// TwinCAT 3 PLC project mobject_graph_vision_pack
// Title: mobject-graph-vision-pack
// Company: mobject
// Author: mobject dev team
// ProjectVersion: 0.7.0
// ProgramVersion: 3.1.4024.0
// libraries:
//   mobject-core,0.5.0,mobject
//   mobject-graph,0.14.0,mobject
//   mobject-graph-plc-pack,0.15.0,mobject
//   Tc2_Standard, * (Beckhoff Automation GmbH)
//   Tc2_System, * (Beckhoff Automation GmbH)
//   Tc2_Utilities, * (Beckhoff Automation GmbH)
//   Tc3_Module, * (Beckhoff Automation GmbH)
//   Tc3_Vision, * (Beckhoff Automation GmbH)
// project tree:
//   Datatypes/Aliases/ _GVCP_REGISTER_ADDRESS.TcPOU, _TcVnMatrix2x3_LREAL.TcPOU (not stored), _TcVnArray4_Point2_REAL.TcPOU, _TcVnArray4_LREAL.TcPOU, _TcVnArray33_UDINT.TcPOU (excluded from build), _TcVnArray10_ITcVnImage.TcPOU, _TcVnArray3_Point2_REAL.TcPOU, _TcVnArray7_LREAL.TcPOU, _TcVnArray8_LREAL.TcPOU, _TcVnMatrix3x3_LREAL.TcPOU, _TcVnPoint.TcPOU, _TcVnPoint2_LREAL.TcPOU, _TcVnPoint3_REAL.TcPOU, _TcVnPoint3_LREAL.TcPOU, _TcVnPoint2_REAL.TcPOU, _TcVnRectangle.TcPOU, _TcVnVector2_DINT.TcPOU, _TcVnPoint2_DINT.TcPOU, _ALIASTYP.TcPOU (excluded from build), _TcVnVector2_INT.TcPOU, _TcVnVector3_SINT.TcPOU, _TcVnVector3_INT.TcPOU, _TcVnVector2_SINT.TcPOU, _TcVnVector2_LREAL.TcPOU, _TcVnVector2_UINT.TcPOU, _TcVnVector2_USINT.TcPOU, _TcVnVector3_UINT.TcPOU, _TcVnVector3_USINT.TcPOU, _TcVnVector4_INT.TcPOU, _TcVnVector4_SINT.TcPOU, _TcVnVector4_LREAL.TcPOU, _TcVnVector3_REAL.TcPOU, _TcVnVector3_LREAL.TcPOU, _TcVnVector2_REAL.TcPOU, _TcVnVector4_DINT.TcPOU, _TcVnVector4_UINT.TcPOU, _TcVnVector4_USINT.TcPOU
//   Datatypes/Arrays/ _Array0to1OfARRAYTYP.TcPOU (excluded from build), _Array0to1OfDINT.TcPOU, _Array0to1OfINT.TcPOU, _Array0to1OfLREAL.TcPOU, _Array0to1OfREAL.TcPOU, _Array0to1OfSINT.TcPOU, _Array0to1OfUINT.TcPOU, _Array0to1OfUSINT.TcPOU, _Array0to1_0to2OfLREAL.TcPOU, _Array0to2_0to2OfLREAL.TcPOU, _Array0to2OfINT.TcPOU, _Array0to2OfLREAL.TcPOU, _Array0to2OfREAL.TcPOU, _Array0to2OfSINT.TcPOU, _Array0to2OfTcVnPoint2_REAL.TcPOU, _Array0to2OfUINT.TcPOU, _Array0to2OfUSINT.TcPOU, _Array0to32OfUDINT.TcPOU, _Array0to3OfDINT.TcPOU, _Array0to3OfINT.TcPOU, _Array0to3OfLREAL.TcPOU, _Array0to3OfSINT.TcPOU, _Array0to3OfTcVnPoint2_REAL.TcPOU, _Array0to3OfUINT.TcPOU, _Array0to3OfUSINT.TcPOU, _Array0to6OfLREAL.TcPOU, _Array0to7OfLREAL.TcPOU, _Array0to9OfITcVnImage.TcPOU
//   Datatypes/Enums/ _ETcVn2dCodeSearchStrategy.TcPOU, _ETcVnAdaptiveThresholdMethod.TcPOU, _ETcVnBarcodeSearchDirection.TcPOU, _ETcVnBarcodeType.TcPOU, _ETcVnBlobCombination.TcPOU, _ETcVnBorderInterpolationMethod.TcPOU, _ETcVnBoostClassifierType.TcPOU (not stored) (excluded from build), _ETcVnCalibrationPattern.TcPOU, _ETcVnCalibrationPatternOrigin.TcPOU, _ETcVnCameraState.TcPOU, _ETcVnClusteringAlgorithm.TcPOU, _ETcVnColorMap.TcPOU, _ETcVnColorMapSize.TcPOU, _ETcVnColorSpaceTransform.TcPOU, _ETcVnColorTrainingMethod.TcPOU, _ETcVnConnectedComponentsAlgorithm.TcPOU, _ETcVnContainerExportFormat.TcPOU, _ETcVnContourApproximationMethod.TcPOU, _ETcVnContourRetrievalMode.TcPOU, _ETcVnContoursMatchComparisonMethod.TcPOU, _ETcVnDiffusivityTypeKAZE.TcPOU, _ETcVnDistanceTransformationLabel.TcPOU, _ETcVnDistanceTransformationMask.TcPOU, _ETcVnDistanceType.TcPOU, _ETcVnDrawMatchesFlags.TcPOU, _ETcVnDrawShape.TcPOU, _ETcVnEdgeDetectionAlgorithm.TcPOU, _ETcVnEdgeDirection.TcPOU, _ETcVnElementType.TcPOU, _ETcVnEstimationAlgorithm.TcPOU, _ETcVnExtremePointDirection.TcPOU, _ETcVnFeatureDescriptorTypeAKAZE.TcPOU, _ETcVnFeatureScalingType.TcPOU (excluded from build), _ETcVnFeatureScoreTypeORB.TcPOU, _ETcVnFilterDirection.TcPOU, _ETcVnFlipAxis.TcPOU, _ETcVnFontType.TcPOU, _ETcVnHoughMethod.TcPOU, _ETcVnInitializableFunction.TcPOU (excluded from build), _ETcVnInterpolationType.TcPOU, _ETcVnKeypointDetectionTypeAGAST.TcPOU, _ETcVnKeypointDetectionTypeFAST.TcPOU, _ETcVnKnn.TcPOU (excluded from build), _ETcVnLineType.TcPOU, _ETcVnMorphologicalOperator.TcPOU, _ETcVnNbc.TcPOU (excluded from build), _ETcVnNormalizationType.TcPOU, _ETcVnOcrModelType.TcPOU (excluded from build), _ETcVnTimestamp.TcPOU (excluded from build), _ETcVnOcrOptions.TcPOU (excluded from build), _ETcVnOrientationMethod.TcPOU, _ETcVnPaddingMode.TcPOU (excluded from build), _ETcVnPixelConnectivity.TcPOU, _ETcVnPixelEncoding.TcPOU, _ETcVnPixelPackMode.TcPOU, _ETcVnPrototypeClusterer.TcPOU (excluded from build), _ETcVnRectangleIntersection.TcPOU, _ETcVnRotationAngle.TcPOU, _ETcVnRTrees.TcPOU (excluded from build), _ETcVnSignedNormalization.TcPOU, _ETcVnSolvePnPMethod.TcPOU (excluded from build), _ETcVnSta.TcPOU (excluded from build), _ETcVnStructuringElementShape.TcPOU, _ETcVnSvm.TcPOU (excluded from build), _ETcVnSvmKernelType.TcPOU (excluded from build), _ETcVnSvmSgdClassifierMarginType.TcPOU (excluded from build), _ETcVnSvmSgdClassifierType.TcPOU (excluded from build), _ETcVnTemplateMatchMethod.TcPOU, _ETcVnThresholdType.TcPOU, _ETcVnVectorCompareMethod.TcPOU, _ETcVnWorldCoordinateSystem.TcPOU, _ETcWatchdogAccumulationType.TcPOU, _GEV_CAMERA_STATE.TcPOU
//   Datatypes/Interfaces/ _ITcVnContainer.TcPOU, _ITcVnImage.TcPOU
//   Datatypes/Structs/ _TcVnDMatch.TcPOU (not stored), _TcVnKeyPoint.TcPOU, _TcVnImageInfo.TcPOU, _TcVnCodeGrades1D.TcPOU (not stored) (excluded from build), _TcVnParamsMSER.TcPOU (not stored), _TcVnParamsKAZE.TcPOU, _TcVnParamsAKAZE.TcPOU (not stored), _TcVnParamsORB.TcPOU, _TcVnParamsSB.TcPOU (not stored), _TcVnParamsBRISK.TcPOU (not stored), _TcVnParamsFAST.TcPOU, _TcVnParamsBlobDetection.TcPOU, _TcVnParamsAGAST.TcPOU, _TcVnCameraCalibrationOptions.TcPOU (not stored), _TcVnParamsGFTT.TcPOU (not stored), _TcVnRotatedRectangle.TcPOU, _TcVnCircularArc.TcPOU, _TcVnSize2_REAL.TcPOU, _TcVnPixelFormat.TcPOU, _TcVnRectangle_DINT.TcPOU, _TcVnRectangle_UDINT.TcPOU
//   Datatypes/ VisionDatatypePack.TcPOU
//   / GVL_COLOURS.TcGVL, VisionPack.TcPOU
//   Nodes/Algebraic Container Operations/ Node_F_VN_AddToContainerElements_DINT.TcPOU, Node_F_VN_AddToContainerElements_INT.TcPOU, Node_F_VN_AddToContainerElements_LREAL.TcPOU, Node_F_VN_AddToContainerElements_REAL.TcPOU, Node_F_VN_AddToContainerElements_SINT.TcPOU (not stored), Node_F_VN_AddToContainerElements_TcVnKeyPoint.TcPOU, Node_F_VN_AddToContainerElements_TcVnPoint2_DINT.TcPOU, Node_F_VN_AddToContainerElements_TcVnPoint2_LREAL.TcPOU, Node_F_VN_AddToContainerElements_TcVnPoint2_REAL.TcPOU, Node_F_VN_AddToContainerElements_TcVnPoint3_LREAL.TcPOU, Node_F_VN_AddToContainerElements_TcVnPoint3_REAL.TcPOU, Node_F_VN_AddToContainerElements_TcVnRectangle_DINT.TcPOU, Node_F_VN_AddToContainerElements_TcVnVector2_DINT.TcPOU, Node_F_VN_AddToContainerElements_TcVnVector2_INT.TcPOU, Node_F_VN_AddToContainerElements_TcVnVector2_REAL.TcPOU, Node_F_VN_AddToContainerElements_TcVnVector2_SINT.TcPOU, Node_F_VN_AddToContainerElements_TcVnVector2_UINT.TcPOU, Node_F_VN_AddToContainerElements_TcVnVector2_USINT.TcPOU, Node_F_VN_AddToContainerElements_TcVnVector3_INT.TcPOU, Node_F_VN_AddToContainerElements_TcVnVector3_REAL.TcPOU, Node_F_VN_AddToContainerElements_TcVnVector3_SINT.TcPOU, Node_F_VN_AddToContainerElements_TcVnVector3_UINT.TcPOU, Node_F_VN_AddToContainerElements_TcVnVector3_USINT.TcPOU, Node_F_VN_AddToContainerElements_TcVnVector4_DINT.TcPOU, Node_F_VN_AddToContainerElements_TcVnVector4_INT.TcPOU, Node_F_VN_AddToContainerElements_TcVnVector4_LREAL.TcPOU, Node_F_VN_AddToContainerElements_TcVnVector4_SINT.TcPOU, Node_F_VN_AddToContainerElements_TcVnVector4_UINT.TcPOU, Node_F_VN_AddToContainerElements_TcVnVector4_USINT.TcPOU, Node_F_VN_AddToContainerElements_UDINT.TcPOU (not stored), Node_F_VN_AddToContainerElements_UINT.TcPOU (not stored), Node_F_VN_AddToContainerElements_ULINT.TcPOU (not stored), Node_F_VN_AddToContainerElements_USINT.TcPOU (not stored)
//   Nodes/Algebraic Image Operations/ Node_F_VN_AddImages.TcPOU (not stored), Node_F_VN_ElementwiseExp.TcPOU, Node_F_VN_ElementwiseLog.TcPOU (not stored), Node_F_VN_MultiplyImageWithScalar.TcPOU (not stored), Node_F_VN_SubtractScalarFromImage.TcPOU (not stored), Node_F_VN_MultiplyImages.TcPOU, Node_F_VN_SubtractImages.TcPOU (not stored), Node_F_VN_MaxImage.TcPOU (not stored), Node_F_VN_BitwiseOrImages.TcPOU (not stored), Node_F_VN_BitwiseNotImage.TcPOU, Node_F_VN_BitwiseAndImages.TcPOU, Node_F_VN_BitwiseXorImages.TcPOU, Node_F_VN_MinImage.TcPOU (not stored), Node_F_VN_DivideImages.TcPOU, Node_F_VN_SubtractImageFromScalar.TcPOU (not stored), Node_F_VN_AddScalarToImage.TcPOU (not stored)
//   Nodes/Basic Container Operations/ Node_F_VN_AppendToContainer_DINT.TcPOU, Node_F_VN_AppendToContainer_INT.TcPOU, Node_F_VN_AppendToContainer_ITcVnContainer.TcPOU, Node_F_VN_AppendToContainer_ITcVnImage.TcPOU, Node_F_VN_AppendToContainer_LREAL.TcPOU, Node_F_VN_AppendToContainer_REAL.TcPOU, Node_F_VN_AppendToContainer_SINT.TcPOU, Node_F_VN_AppendToContainer_TcVnKeyPoint.TcPOU, Node_F_VN_AppendToContainer_TcVnPoint2_DINT.TcPOU, Node_F_VN_AppendToContainer_TcVnPoint2_LREAL.TcPOU, Node_F_VN_AppendToContainer_TcVnPoint2_REAL.TcPOU, Node_F_VN_AppendToContainer_TcVnPoint3_LREAL.TcPOU, Node_F_VN_AppendToContainer_TcVnPoint3_REAL.TcPOU, Node_F_VN_AppendToContainer_TcVnRectangle_DINT.TcPOU, Node_F_VN_AppendToContainer_TcVnDMatch.TcPOU, Node_F_VN_AppendToContainer_TcVnVector2_DINT.TcPOU, Node_F_VN_AppendToContainer_TcVnVector2_INT.TcPOU, Node_F_VN_AppendToContainer_TcVnVector2_REAL.TcPOU, Node_F_VN_AppendToContainer_TcVnVector2_SINT.TcPOU, Node_F_VN_AppendToContainer_TcVnVector2_UINT.TcPOU, Node_F_VN_AppendToContainer_TcVnVector2_USINT.TcPOU, Node_F_VN_AppendToContainer_TcVnVector3_INT.TcPOU, Node_F_VN_AppendToContainer_TcVnVector3_REAL.TcPOU, Node_F_VN_AppendToContainer_TcVnVector3_SINT.TcPOU, Node_F_VN_AppendToContainer_TcVnVector3_UINT.TcPOU, Node_F_VN_AppendToContainer_TcVnVector3_USINT.TcPOU, Node_F_VN_AppendToContainer_TcVnVector4_DINT.TcPOU, Node_F_VN_AppendToContainer_TcVnVector4_INT.TcPOU, Node_F_VN_AppendToContainer_TcVnVector4_LREAL.TcPOU, Node_F_VN_AppendToContainer_TcVnVector4_SINT.TcPOU, Node_F_VN_AppendToContainer_TcVnVector4_UINT.TcPOU, Node_F_VN_AppendToContainer_TcVnVector4_USINT.TcPOU, Node_F_VN_AppendToContainer_UDINT.TcPOU, Node_F_VN_AppendToContainer_UINT.TcPOU, Node_F_VN_AppendToContainer_ULINT.TcPOU, Node_F_VN_AppendToContainer_USINT.TcPOU, Node_F_VN_FillContainerExp_DINT.TcPOU (not stored), Node_F_VN_FillContainerExp_INT.TcPOU, Node_F_VN_FillContainerExp_ITcVnImage.TcPOU, Node_F_VN_FillContainerExp_LREAL.TcPOU (not stored), Node_F_VN_FillContainerExp_REAL.TcPOU (not stored), Node_F_VN_FillContainerExp_SINT.TcPOU, Node_F_VN_FillContainerExp_TcVnDMatch.TcPOU, Node_F_VN_FillContainerExp_TcVnKeyPoint.TcPOU, Node_F_VN_FillContainerExp_TcVnPoint2_DINT.TcPOU, Node_F_VN_FillContainerExp_TcVnPoint2_LREAL.TcPOU, Node_F_VN_FillContainerExp_TcVnPoint2_REAL.TcPOU, Node_F_VN_FillContainerExp_TcVnPoint3_LREAL.TcPOU, Node_F_VN_FillContainerExp_TcVnPoint3_REAL.TcPOU, Node_F_VN_FillContainerExp_TcVnRectangle_DINT.TcPOU, Node_F_VN_FillContainerExp_TcVnVector2_DINT.TcPOU, Node_F_VN_FillContainerExp_TcVnVector2_INT.TcPOU, Node_F_VN_FillContainerExp_TcVnVector2_REAL.TcPOU, Node_F_VN_FillContainerExp_TcVnVector2_SINT.TcPOU, Node_F_VN_FillContainerExp_TcVnVector2_UINT.TcPOU, Node_F_VN_FillContainerExp_TcVnVector2_USINT.TcPOU, Node_F_VN_FillContainerExp_TcVnVector3_INT.TcPOU, Node_F_VN_FillContainerExp_TcVnVector3_REAL.TcPOU, Node_F_VN_FillContainerExp_TcVnVector3_SINT.TcPOU, Node_F_VN_FillContainerExp_TcVnVector3_UINT.TcPOU, Node_F_VN_FillContainerExp_TcVnVector3_USINT.TcPOU, Node_F_VN_FillContainerExp_TcVnVector4_DINT.TcPOU, Node_F_VN_FillContainerExp_TcVnVector4_INT.TcPOU, Node_F_VN_FillContainerExp_TcVnVector4_LREAL.TcPOU, Node_F_VN_FillContainerExp_TcVnVector4_SINT.TcPOU, Node_F_VN_FillContainerExp_TcVnVector4_UINT.TcPOU, Node_F_VN_FillContainerExp_TcVnVector4_USINT.TcPOU, Node_F_VN_FillContainerExp_UDINT.TcPOU, Node_F_VN_FillContainerExp_UINT.TcPOU, Node_F_VN_FillContainerExp_ULINT.TcPOU (not stored), Node_F_VN_FillContainerExp_USINT.TcPOU, Node_F_VN_FillContainer_DINT.TcPOU, Node_F_VN_FillContainer_INT.TcPOU, Node_F_VN_FillContainer_ITcVnImage.TcPOU, Node_F_VN_FillContainer_LREAL.TcPOU, Node_F_VN_FillContainer_REAL.TcPOU, Node_F_VN_FillContainer_SINT.TcPOU, Node_F_VN_FillContainer_TcVnDMatch.TcPOU, Node_F_VN_FillContainer_TcVnKeyPoint.TcPOU, Node_F_VN_FillContainer_TcVnPoint2_DINT.TcPOU, Node_F_VN_FillContainer_TcVnPoint2_LREAL.TcPOU, Node_F_VN_FillContainer_TcVnPoint2_REAL.TcPOU, Node_F_VN_FillContainer_TcVnPoint3_LREAL.TcPOU, Node_F_VN_FillContainer_TcVnPoint3_REAL.TcPOU, Node_F_VN_FillContainer_TcVnRectangle_DINT.TcPOU, Node_F_VN_FillContainer_TcVnVector2_DINT.TcPOU, Node_F_VN_FillContainer_TcVnVector2_INT.TcPOU, Node_F_VN_FillContainer_TcVnVector2_REAL.TcPOU, Node_F_VN_FillContainer_TcVnVector2_SINT.TcPOU, Node_F_VN_FillContainer_TcVnVector2_UINT.TcPOU, Node_F_VN_FillContainer_TcVnVector2_USINT.TcPOU, Node_F_VN_FillContainer_TcVnVector3_INT.TcPOU, Node_F_VN_FillContainer_TcVnVector3_REAL.TcPOU, Node_F_VN_FillContainer_TcVnVector3_SINT.TcPOU, Node_F_VN_FillContainer_TcVnVector3_UINT.TcPOU, Node_F_VN_FillContainer_TcVnVector3_USINT.TcPOU, Node_F_VN_FillContainer_TcVnVector4_DINT.TcPOU, Node_F_VN_FillContainer_TcVnVector4_INT.TcPOU, Node_F_VN_FillContainer_TcVnVector4_LREAL.TcPOU, Node_F_VN_FillContainer_TcVnVector4_SINT.TcPOU, Node_F_VN_FillContainer_TcVnVector4_UINT.TcPOU, Node_F_VN_FillContainer_TcVnVector4_USINT.TcPOU, Node_F_VN_FillContainer_UDINT.TcPOU, Node_F_VN_FillContainer_UINT.TcPOU, Node_F_VN_FillContainer_ULINT.TcPOU, Node_F_VN_FillContainer_USINT.TcPOU, Node_F_VN_GetAt_DINT.TcPOU (not stored), Node_F_VN_GetAt_INT.TcPOU, Node_F_VN_GetAt_ITcVnContainer.TcPOU (not stored), Node_F_VN_GetAt_ITcVnImage.TcPOU, Node_F_VN_GetAt_LREAL.TcPOU, Node_F_VN_GetAt_REAL.TcPOU (not stored), Node_F_VN_GetAt_SINT.TcPOU (not stored), Node_F_VN_GetAt_TcVnDMatch.TcPOU, Node_F_VN_GetAt_TcVnKeyPoint.TcPOU, Node_F_VN_GetAt_TcVnPoint2_DINT.TcPOU, Node_F_VN_GetAt_TcVnPoint2_LREAL.TcPOU, Node_F_VN_GetAt_TcVnPoint2_REAL.TcPOU, Node_F_VN_GetAt_TcVnPoint3_LREAL.TcPOU, Node_F_VN_GetAt_TcVnPoint3_REAL.TcPOU, Node_F_VN_GetAt_TcVnRectangle_DINT.TcPOU, Node_F_VN_GetAt_TcVnVector2_DINT.TcPOU, Node_F_VN_GetAt_TcVnVector2_INT.TcPOU, Node_F_VN_GetAt_TcVnVector2_REAL.TcPOU, Node_F_VN_GetAt_TcVnVector2_SINT.TcPOU, Node_F_VN_GetAt_TcVnVector2_UINT.TcPOU, Node_F_VN_GetAt_TcVnVector2_USINT.TcPOU, Node_F_VN_GetAt_TcVnVector3_INT.TcPOU, Node_F_VN_GetAt_TcVnVector3_REAL.TcPOU, Node_F_VN_GetAt_TcVnVector3_SINT.TcPOU, Node_F_VN_GetAt_TcVnVector3_UINT.TcPOU, Node_F_VN_GetAt_TcVnVector3_USINT.TcPOU, Node_F_VN_GetAt_TcVnVector4_DINT.TcPOU, Node_F_VN_GetAt_TcVnVector4_INT.TcPOU, Node_F_VN_GetAt_TcVnVector4_LREAL.TcPOU, Node_F_VN_GetAt_TcVnVector4_SINT.TcPOU, Node_F_VN_GetAt_TcVnVector4_UINT.TcPOU, Node_F_VN_GetAt_TcVnVector4_USINT.TcPOU, Node_F_VN_GetAt_UDINT.TcPOU, Node_F_VN_GetAt_UINT.TcPOU (not stored), Node_F_VN_GetAt_ULINT.TcPOU (not stored), Node_F_VN_GetAt_USINT.TcPOU (not stored), Node_F_VN_GetNumberOfElements.TcPOU, Node_F_VN_InsertIntoContainer_DINT.TcPOU, Node_F_VN_InsertIntoContainer_INT.TcPOU, Node_F_VN_InsertIntoContainer_ITcVnContainer.TcPOU, Node_F_VN_InsertIntoContainer_ITcVnImage.TcPOU, Node_F_VN_InsertIntoContainer_LREAL.TcPOU, Node_F_VN_InsertIntoContainer_REAL.TcPOU, Node_F_VN_InsertIntoContainer_SINT.TcPOU, Node_F_VN_InsertIntoContainer_TcVnDMatch.TcPOU, Node_F_VN_InsertIntoContainer_TcVnKeyPoint.TcPOU, Node_F_VN_InsertIntoContainer_TcVnPoint2_DINT.TcPOU, Node_F_VN_InsertIntoContainer_TcVnPoint2_LREAL.TcPOU, Node_F_VN_InsertIntoContainer_TcVnPoint2_REAL.TcPOU, Node_F_VN_InsertIntoContainer_TcVnPoint3_LREAL.TcPOU, Node_F_VN_InsertIntoContainer_TcVnPoint3_REAL.TcPOU, Node_F_VN_InsertIntoContainer_TcVnRectangle_DINT.TcPOU, Node_F_VN_InsertIntoContainer_TcVnVector2_DINT.TcPOU, Node_F_VN_InsertIntoContainer_TcVnVector2_INT.TcPOU, Node_F_VN_InsertIntoContainer_TcVnVector2_REAL.TcPOU, Node_F_VN_InsertIntoContainer_TcVnVector2_SINT.TcPOU, Node_F_VN_InsertIntoContainer_TcVnVector2_UINT.TcPOU, Node_F_VN_InsertIntoContainer_TcVnVector2_USINT.TcPOU, Node_F_VN_InsertIntoContainer_TcVnVector3_INT.TcPOU, Node_F_VN_InsertIntoContainer_TcVnVector3_REAL.TcPOU, Node_F_VN_InsertIntoContainer_TcVnVector3_SINT.TcPOU, Node_F_VN_InsertIntoContainer_TcVnVector3_UINT.TcPOU, Node_F_VN_InsertIntoContainer_TcVnVector3_USINT.TcPOU, Node_F_VN_InsertIntoContainer_TcVnVector4_DINT.TcPOU, Node_F_VN_InsertIntoContainer_TcVnVector4_INT.TcPOU, Node_F_VN_InsertIntoContainer_TcVnVector4_LREAL.TcPOU, Node_F_VN_InsertIntoContainer_TcVnVector4_SINT.TcPOU, Node_F_VN_InsertIntoContainer_TcVnVector4_UINT.TcPOU, Node_F_VN_InsertIntoContainer_TcVnVector4_USINT.TcPOU, Node_F_VN_InsertIntoContainer_UDINT.TcPOU, Node_F_VN_InsertIntoContainer_UINT.TcPOU, Node_F_VN_InsertIntoContainer_ULINT.TcPOU, Node_F_VN_InsertIntoContainer_USINT.TcPOU, Node_F_VN_SetAt_DINT.TcPOU, Node_F_VN_SetAt_INT.TcPOU, Node_F_VN_SetAt_ITcVnContainer.TcPOU, Node_F_VN_SetAt_ITcVnImage.TcPOU, Node_F_VN_SetAt_LREAL.TcPOU, Node_F_VN_SetAt_REAL.TcPOU, Node_F_VN_SetAt_SINT.TcPOU, Node_F_VN_SetAt_TcVnDMatch.TcPOU, Node_F_VN_SetAt_TcVnKeyPoint.TcPOU, Node_F_VN_SetAt_TcVnPoint2_DINT.TcPOU, Node_F_VN_SetAt_TcVnPoint2_LREAL.TcPOU, Node_F_VN_SetAt_TcVnPoint2_REAL.TcPOU, Node_F_VN_SetAt_TcVnPoint3_LREAL.TcPOU, Node_F_VN_SetAt_TcVnPoint3_REAL.TcPOU, Node_F_VN_SetAt_TcVnRectangle_DINT.TcPOU, Node_F_VN_SetAt_TcVnVector2_DINT.TcPOU, Node_F_VN_SetAt_TcVnVector2_INT.TcPOU, Node_F_VN_SetAt_TcVnVector2_REAL.TcPOU, Node_F_VN_SetAt_TcVnVector2_SINT.TcPOU, Node_F_VN_SetAt_TcVnVector2_UINT.TcPOU, Node_F_VN_SetAt_TcVnVector2_USINT.TcPOU, Node_F_VN_SetAt_TcVnVector3_INT.TcPOU, Node_F_VN_SetAt_TcVnVector3_REAL.TcPOU, Node_F_VN_SetAt_TcVnVector3_SINT.TcPOU, Node_F_VN_SetAt_TcVnVector3_UINT.TcPOU, Node_F_VN_SetAt_TcVnVector3_USINT.TcPOU, Node_F_VN_SetAt_TcVnVector4_DINT.TcPOU, Node_F_VN_SetAt_TcVnVector4_INT.TcPOU, Node_F_VN_SetAt_TcVnVector4_LREAL.TcPOU, Node_F_VN_SetAt_TcVnVector4_SINT.TcPOU, Node_F_VN_SetAt_TcVnVector4_UINT.TcPOU, Node_F_VN_SetAt_TcVnVector4_USINT.TcPOU, Node_F_VN_SetAt_UDINT.TcPOU, Node_F_VN_SetAt_UINT.TcPOU, Node_F_VN_SetAt_ULINT.TcPOU, Node_F_VN_SetAt_USINT.TcPOU
//   Nodes/Basic Image Operations/ Node_F_VN_ConvertElementType.TcPOU, Node_F_VN_ConvertElementTypeExp.TcPOU (not stored), Node_F_VN_CopyImage.TcPOU, Node_F_VN_GetPixelFormat.TcPOU, Node_F_VN_ResetRoi.TcPOU (not stored), Node_F_VN_SetRoi.TcPOU (not stored), Node_F_VN_GetImageChannel.TcPOU (not stored), Node_F_VN_GetImageHeight.TcPOU, Node_F_VN_GetImageWidth.TcPOU, Node_F_VN_GetImageInfo.TcPOU, Node_F_VN_GetRoi.TcPOU (not stored), Node_F_VN_SetRoi_TcVnRectangle_DINT.TcPOU (excluded from build)
//   Nodes/Code Reading/ Node_F_VN_ReadQRCode.TcPOU (not stored), Node_F_VN_ReadDataMatrixCode.TcPOU
//   Nodes/Constants/ Node_RGBA_BLUE.TcPOU, Node_RGBA_MAGENTA.TcPOU, Node_RGBA_CYAN.TcPOU, Node_RGBA_YELLOW.TcPOU, Node_RGBA_WHITE.TcPOU, Node_RGBA_RED.TcPOU (not stored), Node_RGBA_GREEN.TcPOU (not stored), Node_RGBA_BLACK.TcPOU (not stored)
//   Nodes/Container Statistics/ Node_F_VN_MaxElementElementwise_DINT.TcPOU, Node_F_VN_MaxElementElementwise_INT.TcPOU, Node_F_VN_MaxElementElementwise_LREAL.TcPOU, Node_F_VN_MaxElementElementwise_REAL.TcPOU, Node_F_VN_MaxElementElementwise_SINT.TcPOU, Node_F_VN_MaxElementElementwise_TcVnPoint2_DINT.TcPOU, Node_F_VN_MaxElementElementwise_TcVnPoint2_LREAL.TcPOU (not stored), Node_F_VN_MaxElementElementwise_TcVnPoint2_REAL.TcPOU (not stored), Node_F_VN_MaxElementElementwise_TcVnPoint3_LREAL.TcPOU (not stored), Node_F_VN_MaxElementElementwise_TcVnPoint3_REAL.TcPOU (not stored), Node_F_VN_MaxElementElementwise_TcVnVector2_DINT.TcPOU (not stored), Node_F_VN_MaxElementElementwise_TcVnVector2_INT.TcPOU (not stored), Node_F_VN_MaxElementElementwise_TcVnVector2_REAL.TcPOU, Node_F_VN_MaxElementElementwise_TcVnVector2_SINT.TcPOU, Node_F_VN_MaxElementElementwise_TcVnVector2_UINT.TcPOU (not stored), Node_F_VN_MaxElementElementwise_TcVnVector2_USINT.TcPOU (not stored), Node_F_VN_MaxElementElementwise_TcVnVector3_INT.TcPOU, Node_F_VN_MaxElementElementwise_TcVnVector3_REAL.TcPOU (not stored), Node_F_VN_MaxElementElementwise_TcVnVector3_SINT.TcPOU, Node_F_VN_MaxElementElementwise_TcVnVector3_UINT.TcPOU (not stored), Node_F_VN_MaxElementElementwise_TcVnVector3_USINT.TcPOU (not stored), Node_F_VN_MaxElementElementwise_TcVnVector4_DINT.TcPOU (not stored), Node_F_VN_MaxElementElementwise_TcVnVector4_INT.TcPOU, Node_F_VN_MaxElementElementwise_TcVnVector4_LREAL.TcPOU (not stored), Node_F_VN_MaxElementElementwise_TcVnVector4_SINT.TcPOU, Node_F_VN_MaxElementElementwise_TcVnVector4_UINT.TcPOU, Node_F_VN_MaxElementElementwise_TcVnVector4_USINT.TcPOU, Node_F_VN_MaxElementElementwise_UDINT.TcPOU, Node_F_VN_MaxElementElementwise_UINT.TcPOU, Node_F_VN_MaxElementElementwise_ULINT.TcPOU, Node_F_VN_MaxElementElementwise_USINT.TcPOU, Node_F_VN_MedianElementElementwise_DINT.TcPOU, Node_F_VN_MedianElementElementwise_INT.TcPOU, Node_F_VN_MedianElementElementwise_LREAL.TcPOU, Node_F_VN_MedianElementElementwise_REAL.TcPOU, Node_F_VN_MedianElementElementwise_SINT.TcPOU, Node_F_VN_MedianElementElementwise_TcVnPoint2_DINT.TcPOU, Node_F_VN_MedianElementElementwise_TcVnPoint2_LREAL.TcPOU, Node_F_VN_MedianElementElementwise_TcVnPoint2_REAL.TcPOU, Node_F_VN_MedianElementElementwise_TcVnPoint3_LREAL.TcPOU, Node_F_VN_MedianElementElementwise_TcVnPoint3_REAL.TcPOU, Node_F_VN_MedianElementElementwise_TcVnVector2_DINT.TcPOU, Node_F_VN_MedianElementElementwise_TcVnVector2_INT.TcPOU, Node_F_VN_MedianElementElementwise_TcVnVector2_REAL.TcPOU, Node_F_VN_MedianElementElementwise_TcVnVector2_SINT.TcPOU, Node_F_VN_MedianElementElementwise_TcVnVector2_UINT.TcPOU, Node_F_VN_MedianElementElementwise_TcVnVector2_USINT.TcPOU, Node_F_VN_MedianElementElementwise_TcVnVector3_INT.TcPOU, Node_F_VN_MedianElementElementwise_TcVnVector3_REAL.TcPOU, Node_F_VN_MedianElementElementwise_TcVnVector3_SINT.TcPOU, Node_F_VN_MedianElementElementwise_TcVnVector3_UINT.TcPOU, Node_F_VN_MedianElementElementwise_TcVnVector3_USINT.TcPOU, Node_F_VN_MedianElementElementwise_TcVnVector4_DINT.TcPOU, Node_F_VN_MedianElementElementwise_TcVnVector4_INT.TcPOU, Node_F_VN_MedianElementElementwise_TcVnVector4_LREAL.TcPOU, Node_F_VN_MedianElementElementwise_TcVnVector4_SINT.TcPOU, Node_F_VN_MedianElementElementwise_TcVnVector4_UINT.TcPOU, Node_F_VN_MedianElementElementwise_TcVnVector4_USINT.TcPOU, Node_F_VN_MedianElementElementwise_UDINT.TcPOU, Node_F_VN_MedianElementElementwise_UINT.TcPOU, Node_F_VN_MedianElementElementwise_ULINT.TcPOU, Node_F_VN_MedianElementElementwise_USINT.TcPOU, Node_F_VN_MinElementElementwise_DINT.TcPOU, Node_F_VN_MinElementElementwise_INT.TcPOU, Node_F_VN_MinElementElementwise_LREAL.TcPOU, Node_F_VN_MinElementElementwise_REAL.TcPOU, Node_F_VN_MinElementElementwise_SINT.TcPOU, Node_F_VN_MinElementElementwise_TcVnPoint2_DINT.TcPOU, Node_F_VN_MinElementElementwise_TcVnPoint2_LREAL.TcPOU, Node_F_VN_MinElementElementwise_TcVnPoint2_REAL.TcPOU, Node_F_VN_MinElementElementwise_TcVnPoint3_LREAL.TcPOU, Node_F_VN_MinElementElementwise_TcVnPoint3_REAL.TcPOU, Node_F_VN_MinElementElementwise_TcVnVector2_DINT.TcPOU, Node_F_VN_MinElementElementwise_TcVnVector2_INT.TcPOU, Node_F_VN_MinElementElementwise_TcVnVector2_REAL.TcPOU, Node_F_VN_MinElementElementwise_TcVnVector2_SINT.TcPOU, Node_F_VN_MinElementElementwise_TcVnVector2_UINT.TcPOU, Node_F_VN_MinElementElementwise_TcVnVector2_USINT.TcPOU, Node_F_VN_MinElementElementwise_TcVnVector3_INT.TcPOU, Node_F_VN_MinElementElementwise_TcVnVector3_REAL.TcPOU, Node_F_VN_MinElementElementwise_TcVnVector3_SINT.TcPOU, Node_F_VN_MinElementElementwise_TcVnVector3_UINT.TcPOU, Node_F_VN_MinElementElementwise_TcVnVector3_USINT.TcPOU, Node_F_VN_MinElementElementwise_TcVnVector4_DINT.TcPOU, Node_F_VN_MinElementElementwise_TcVnVector4_INT.TcPOU, Node_F_VN_MinElementElementwise_TcVnVector4_LREAL.TcPOU, Node_F_VN_MinElementElementwise_TcVnVector4_SINT.TcPOU, Node_F_VN_MinElementElementwise_TcVnVector4_UINT.TcPOU, Node_F_VN_MinElementElementwise_TcVnVector4_USINT.TcPOU, Node_F_VN_MinElementElementwise_UDINT.TcPOU, Node_F_VN_MinElementElementwise_UINT.TcPOU, Node_F_VN_MinElementElementwise_ULINT.TcPOU, Node_F_VN_MinElementElementwise_USINT.TcPOU
//   Nodes/Contour Analysis/ Node_F_VN_FitLine.TcPOU
//   Nodes/Drawing/ Node_F_VN_DrawContours.TcPOU, Node_F_VN_DrawLine.TcPOU, Node_F_VN_DrawCircle.TcPOU (not stored), Node_F_VN_DrawLine_TcVnVector4_LREAL.TcPOU, Node_F_VN_PutLabel.TcPOU, Node_F_VN_PutText.TcPOU
//   Nodes/Geometric and Coordinate Transformations/ Node_F_VN_PyramidDown.TcPOU (not stored), Node_F_VN_FlipImage.TcPOU, Node_F_VN_PyramidUp.TcPOU (not stored)
//   Nodes/Image Analysis/ Node_F_VN_CountNonZeroPixels.TcPOU
//   Nodes/Image Analysis/Object Detection/ Node_F_VN_DetectBlobs.TcPOU
//   Nodes/Image Color and Contrast Processing/ Node_F_VN_ApplyColorMap.TcPOU, Node_F_VN_InvertImageColor.TcPOU (not stored), Node_F_VN_ConvertColorSpace.TcPOU, Node_F_VN_GenerateColorMap.TcPOU, Node_F_VN_NormalizeImage.TcPOU (not stored)
//   Nodes/Image Filtering/ Node_F_VN_LocalMaxima.TcPOU, Node_F_VN_DarkBorderObjects.TcPOU (not stored), Node_F_VN_FillHoles.TcPOU (not stored), Node_F_VN_BoxFilter.TcPOU, Node_F_VN_BrightBorderObjects.TcPOU (not stored), Node_F_VN_GaussianFilter.TcPOU, Node_F_VN_LaplacianFilter.TcPOU, Node_F_VN_LocalMinima.TcPOU (not stored)
//   Nodes/Image Segmentation/ Node_F_VN_Threshold.TcPOU
//   Nodes/Keypoint Features/ Node_F_VN_KeyPointsAGAST.TcPOU (not stored), Node_F_VN_KeyPointsGFTT.TcPOU (not stored), Node_F_VN_KeyPointsFAST.TcPOU (not stored), Node_F_VN_KeyPointsMSER.TcPOU, Node_F_VN_KeyPointsSB.TcPOU (not stored)
//   Nodes/Measurement/ Node_F_VN_LocateEdge.TcPOU, Node_F_VN_LocateEdges.TcPOU (not stored), Node_F_VN_LocateEdgeExp.TcPOU (not stored), Node_F_VN_LocateEdgesExp.TcPOU (not stored), Node_F_VN_LocateEllipse.TcPOU (not stored)
//   Nodes/ VisionNodePack.TcPOU
//   Nodes/VisionNode/ VisionNode.TcPOU (not stored)

// ---- GVL_COLOURS.TcGVL
{attribute 'qualified_only'}
VAR_GLOBAL
    RGBA_BLACK   : TcVnVector4_LREAL := [0, 0, 0, 255];
    RGBA_RED     : TcVnVector4_LREAL := [255, 0, 0, 255];
    RGBA_YELLOW  : TcVnVector4_LREAL := [255, 255, 0, 255];
    RGBA_GREEN   : TcVnVector4_LREAL := [0, 255, 0, 255];
    RGBA_CYAN    : TcVnVector4_LREAL := [0, 255, 255, 255];
    RGBA_BLUE    : TcVnVector4_LREAL := [0, 0, 255, 255];
    RGBA_MAGENTA : TcVnVector4_LREAL := [255, 0, 255, 255];
    RGBA_WHITE   : TcVnVector4_LREAL := [255, 255, 255, 255];
END_VAR

// ---- Datatypes/Aliases/_GVCP_REGISTER_ADDRESS.TcPOU
{attribute 'linkalways'} 
{attribute 'no_explicit_call' := 'This FB is a CLASS and must be accessed using methods or properties'}
{attribute 'enable_dynamic_creation'}
FUNCTION_BLOCK _GVCP_REGISTER_ADDRESS EXTENDS AliasDatatypeBase
VAR
	localData : GVCP_REGISTER_ADDRESS;
	activeData : REFERENCE TO GVCP_REGISTER_ADDRESS REF= localData;
	aliasBaseDatatype : _UDINT(0);
END_VAR

PROPERTY PUBLIC Address : PVOID
GET
Address := ADR(activeData);
END_GET
END_PROPERTY

METHOD PUBLIC ClearReference
VAR_INPUT
END_VAR
activeData REF= localData;
SetBaseDatatypeReference();
END_METHOD

METHOD PUBLIC Clone : I_Datatype
VAR
    pClone : POINTER TO _GVCP_REGISTER_ADDRESS;
END_VAR
pClone := __NEW(_GVCP_REGISTER_ADDRESS);
Clone := pClone^;
END_METHOD

METHOD FB_init : BOOL
VAR_INPUT
	bInitRetains : BOOL; // if TRUE, the retain variables are initialized (warm start / cold start)
	bInCopyCode : BOOL;  // if TRUE, the instance afterwards gets moved into the copy code (online change)
	//InitialValue : TcVnArray33_UDINT; // if possible, not all values can be initialized
END_VAR
//localData := InitialValue; // if possible, not all values can be initialized
SetBaseDatatypeReference();
AddBaseDatatype(aliasBaseDatatype);
END_METHOD

PROPERTY PUBLIC Identifier : T_MAXSTRING
GET
Identifier := 'GVCP_REGISTER_ADDRESS';
END_GET
END_PROPERTY

METHOD PUBLIC MakeReferenceTo
VAR_INPUT
	ReferenceTarget : REFERENCE TO GVCP_REGISTER_ADDRESS;
END_VAR
activeData REF= ReferenceTarget;
SetBaseDatatypeReference();
END_METHOD

METHOD PROTECTED SetBaseDatatypeReference
VAR_INPUT
END_VAR
aliasBaseDatatype.MakeReferenceTo(activeData);
END_METHOD

PROPERTY PUBLIC Size : UDINT
GET
Size := SIZEOF(activeData);
END_GET
END_PROPERTY

METHOD TryMakeReferenceTo : BOOL
VAR_INPUT
	Target : I_Datatype;
END_VAR
VAR
	targetAsAlias : I_AliasDatatype;
	pTargetData : POINTER TO GVCP_REGISTER_ADDRESS;
END_VAR
IF NOT Target.TryResolveAsAliasDatatype(targetAsAlias) THEN
	RETURN;
END_IF

IF targetAsAlias.Identifier <> Identifier THEN
	RETURN;
END_IF

pTargetData := Target.Address;
activeData REF= pTargetData^;
SetBaseDatatypeReference();
TryMakeReferenceTo := TRUE;
END_METHOD

PROPERTY PUBLIC Value : REFERENCE TO GVCP_REGISTER_ADDRESS
GET
Value REF= activeData;
END_GET
END_PROPERTY

END_FUNCTION_BLOCK

// ---- Datatypes/Aliases/_TcVnArray4_Point2_REAL.TcPOU
{attribute 'linkalways'} 
{attribute 'no_explicit_call' := 'This FB is a CLASS and must be accessed using methods or properties'}
{attribute 'enable_dynamic_creation'}
FUNCTION_BLOCK _TcVnArray4_Point2_REAL EXTENDS AliasDatatypeBase
VAR
	localData : TcVnArray4_Point2_REAL;
	activeData : REFERENCE TO TcVnArray4_Point2_REAL REF= localData;
	aliasBaseDatatype : _Array0to3OfTcVnPoint2_REAL;
END_VAR

PROPERTY PUBLIC Address : PVOID
GET
Address := ADR(activeData);
END_GET
END_PROPERTY

METHOD PUBLIC ClearReference
VAR_INPUT
END_VAR
activeData REF= localData;
SetBaseDatatypeReference();
END_METHOD

METHOD PUBLIC Clone : I_Datatype
VAR
    pClone : POINTER TO _TcVnArray4_Point2_REAL;
END_VAR
pClone := __NEW(_TcVnArray4_Point2_REAL);
Clone := pClone^;
END_METHOD

METHOD FB_init : BOOL
VAR_INPUT
	bInitRetains : BOOL; // if TRUE, the retain variables are initialized (warm start / cold start)
	bInCopyCode : BOOL;  // if TRUE, the instance afterwards gets moved into the copy code (online change)
	//InitialValue : TcVnArray4_LREAL; // if possible, not all values can be initialized
END_VAR
//localData := InitialValue; // if possible, not all values can be initialized
SetBaseDatatypeReference();
AddBaseDatatype(aliasBaseDatatype);
END_METHOD

PROPERTY PUBLIC Identifier : T_MAXSTRING
GET
Identifier := 'TcVnArray4_Point2_REAL';
END_GET
END_PROPERTY

METHOD PUBLIC MakeReferenceTo
VAR_INPUT
	ReferenceTarget : REFERENCE TO TcVnArray4_Point2_REAL;
END_VAR
activeData REF= ReferenceTarget;
SetBaseDatatypeReference();
END_METHOD

METHOD PROTECTED SetBaseDatatypeReference
VAR_INPUT
END_VAR
aliasBaseDatatype.MakeReferenceTo(activeData);
END_METHOD

PROPERTY PUBLIC Size : UDINT
GET
Size := SIZEOF(activeData);
END_GET
END_PROPERTY

METHOD TryMakeReferenceTo : BOOL
VAR_INPUT
	Target : I_Datatype;
END_VAR
VAR
	pTargetData : POINTER TO TcVnArray4_Point2_REAL;
END_VAR
IF NOT IsEquivalentTo(Target) THEN
	RETURN;
END_IF

pTargetData := Target.Address;
activeData REF= pTargetData^;
SetBaseDatatypeReference();
TryMakeReferenceTo := TRUE;
END_METHOD

PROPERTY PUBLIC Value : REFERENCE TO TcVnArray4_Point2_REAL
GET
Value REF= activeData;
END_GET
END_PROPERTY

END_FUNCTION_BLOCK

// ---- Datatypes/Arrays/_Array0to3OfTcVnPoint2_REAL.TcPOU
{attribute 'linkalways'} 
{attribute 'no_explicit_call' := 'This FB is a CLASS and must be accessed using methods or properties'}
{attribute 'enable_dynamic_creation'}
FUNCTION_BLOCK _Array0to3OfTcVnPoint2_REAL EXTENDS ArrayDatatypeBase_1D
VAR CONSTANT
	lBound : DINT := 0;
	uBound : DINT := 3;
END_VAR
VAR
	localData : ARRAY [lBound..uBound] OF TcVnPoint2_REAL;
	activeData : REFERENCE TO ARRAY [lBound..uBound] OF TcVnPoint2_REAL REF= localData;
	elements : ARRAY [lBound..uBound] OF _TcVnPoint2_REAL;
	baseType : _TcVnPoint2_REAL;
END_VAR

PROPERTY PUBLIC Address : PVOID
GET
Address := ADR(activeData);
END_GET
END_PROPERTY

PROPERTY PUBLIC BaseDatatype : I_Datatype
GET
BaseDatatype := baseType;
END_GET
END_PROPERTY

METHOD PUBLIC ClearReference
VAR_INPUT
END_VAR
activeData REF= localData;
SetElementReference();
END_METHOD

METHOD PUBLIC Clone : I_Datatype
VAR
    pClone : POINTER TO _Array0to3OfTcVnPoint2_REAL;
END_VAR
pClone := __NEW(_Array0to3OfTcVnPoint2_REAL());
pClone^.Value := Value;
Clone := pClone^;
END_METHOD

METHOD FB_init : BOOL
VAR_INPUT
	bInitRetains : BOOL; // if TRUE, the retain variables are initialized (warm start / cold start)
	bInCopyCode : BOOL;  // if TRUE, the instance afterwards gets moved into the copy code (online change)
END_VAR
SetElementReference();
END_METHOD

METHOD PUBLIC MakeReferenceTo
VAR_INPUT
	ReferenceTarget : REFERENCE TO ARRAY [lBound..uBound] OF TcVnPoint2_REAL;
END_VAR
activeData REF= ReferenceTarget;
SetElementReference();
END_METHOD

METHOD PROTECTED OnSerializeArrayValues
VAR_INPUT
	Serializer : I_Serializer;
END_VAR
VAR
	i : DINT;
END_VAR
FOR i := lBound TO uBound DO
	elements[i].SerializeWith(Serializer);
END_FOR
END_METHOD

METHOD PROTECTED SetElementReference
VAR_INPUT
END_VAR
VAR
	i : DINT;
END_VAR
FOR i := lBound TO uBound DO
	elements[i].MakeReferenceTo(activeData[i]);
END_FOR
END_METHOD

PROPERTY PUBLIC Size : UDINT
GET
Size := SIZEOF(activeData);
END_GET
END_PROPERTY

METHOD PROTECTED TryDeserializeArrayValues : BOOL
VAR_INPUT
	Deserializer : I_Deserializer;
	Feedback : I_DeserializerFeedback;
END_VAR
VAR
	enumerator : I_DeserializerArrayForwardEnumerator;
	i : DINT;
END_VAR
enumerator := Deserializer.GetArrayEnumerator();
i := lBound;

WHILE enumerator.MoveNext() AND i <= uBound DO
	
	IF NOT elements[i].TryDeserializeFrom(enumerator.Current, Feedback) THEN
		EXIT;
	END_IF
	i := i + 1;

END_WHILE
enumerator.Dispose();
END_METHOD

METHOD PUBLIC TryGetElementAsDatatypeByIndex : BOOL
VAR_INPUT
	Index : DINT;
	Destination : REFERENCE TO I_Datatype;
END_VAR
IF Index < lbound OR Index > ubound THEN
	RETURN;
END_IF

Destination := elements[Index];
TryGetElementAsDatatypeByIndex := TRUE;
END_METHOD

METHOD PUBLIC TryGetLowerBound : BOOL
VAR_INPUT
	Dimention : UDINT;
	Destination : REFERENCE TO DINT;
END_VAR
IF Dimention = 1 THEN
	Destination := lBound;
	TryGetLowerBound := TRUE;
END_IF
END_METHOD

METHOD PUBLIC TryGetUpperBound : BOOL
VAR_INPUT
	Dimention : UDINT;
	Destination : REFERENCE TO DINT;
END_VAR
IF Dimention = 1 THEN
	Destination := uBound;
	TryGetUpperBound := TRUE;
END_IF
END_METHOD

METHOD TryMakeReferenceTo : BOOL
VAR_INPUT
	Target : I_Datatype;
END_VAR
VAR
	targetAsArray : I_ArrayDatatype;
	pTargetData : POINTER TO ARRAY [lBound..uBound] OF TcVnPoint2_REAL;
END_VAR
IF NOT Target.TryResolveAsArrayDatatype(targetAsArray) THEN
	RETURN;
END_IF

IF NOT (targetAsArray.Identifier = Identifier) THEN
	RETURN;
END_IF

pTargetData := Target.Address;
activeData REF= pTargetData^;
SetElementReference();
TryMakeReferenceTo := TRUE;
END_METHOD

PROPERTY PUBLIC Value : REFERENCE TO ARRAY [lBound..uBound] OF TcVnPoint2_REAL;
GET
Value ref= activeData;
END_GET
END_PROPERTY

END_FUNCTION_BLOCK

// ---- Datatypes/Aliases/_TcVnPoint2_REAL.TcPOU
{attribute 'linkalways'} 
{attribute 'no_explicit_call' := 'This FB is a CLASS and must be accessed using methods or properties'}
{attribute 'enable_dynamic_creation'}
FUNCTION_BLOCK _TcVnPoint2_REAL EXTENDS AliasDatatypeBase
VAR
	localData : TcVnPoint2_REAL;
	activeData : REFERENCE TO TcVnPoint2_REAL REF= localData;
	aliasBaseDatatype : _TcVnVector2_REAL;
END_VAR

PROPERTY PUBLIC Address : PVOID
GET
Address := ADR(activeData);
END_GET
END_PROPERTY

METHOD PUBLIC ClearReference
VAR_INPUT
END_VAR
activeData REF= localData;
SetBaseDatatypeReference();
END_METHOD

METHOD PUBLIC Clone : I_Datatype
VAR
    pClone : POINTER TO _TcVnPoint2_REAL;
END_VAR
pClone := __NEW(_TcVnPoint2_REAL);
Clone := pClone^;
END_METHOD

METHOD FB_init : BOOL
VAR_INPUT
	bInitRetains : BOOL; // if TRUE, the retain variables are initialized (warm start / cold start)
	bInCopyCode : BOOL;  // if TRUE, the instance afterwards gets moved into the copy code (online change)
	//InitialValue : <type>; // if possible, not all values can be initialized
END_VAR
//localData := InitialValue; // if possible, not all values can be initialized
SetBaseDatatypeReference();
AddBaseDatatype(aliasBaseDatatype);
END_METHOD

PROPERTY PUBLIC Identifier : T_MAXSTRING
GET
Identifier := 'TcVnPoint2_REAL';
END_GET
END_PROPERTY

METHOD PUBLIC MakeReferenceTo
VAR_INPUT
	ReferenceTarget : REFERENCE TO TcVnPoint2_REAL;
END_VAR
activeData REF= ReferenceTarget;
SetBaseDatatypeReference();
END_METHOD

METHOD PROTECTED SetBaseDatatypeReference
VAR_INPUT
END_VAR
aliasBaseDatatype.MakeReferenceTo(activeData);
END_METHOD

PROPERTY PUBLIC Size : UDINT
GET
Size := SIZEOF(activeData);
END_GET
END_PROPERTY

METHOD TryMakeReferenceTo : BOOL
VAR_INPUT
	Target : I_Datatype;
END_VAR
VAR
	pTargetData : POINTER TO TcVnPoint2_REAL;
END_VAR
IF NOT IsEquivalentTo(Target) THEN
	RETURN;
END_IF

pTargetData := Target.Address;
activeData REF= pTargetData^;
SetBaseDatatypeReference();
TryMakeReferenceTo := TRUE;
END_METHOD

PROPERTY PUBLIC Value : REFERENCE TO TcVnPoint2_REAL
GET
Value REF= activeData;
END_GET
END_PROPERTY

END_FUNCTION_BLOCK

// ---- Datatypes/Aliases/_TcVnVector2_REAL.TcPOU
{attribute 'linkalways'} 
{attribute 'no_explicit_call' := 'This FB is a CLASS and must be accessed using methods or properties'}
{attribute 'enable_dynamic_creation'}
FUNCTION_BLOCK _TcVnVector2_REAL EXTENDS AliasDatatypeBase
VAR
	localData : TcVnVector2_REAL;
	activeData : REFERENCE TO TcVnVector2_REAL REF= localData;
	aliasBaseDatatype : _Array0to1OfREAL;
END_VAR

PROPERTY PUBLIC Address : PVOID
GET
Address := ADR(activeData);
END_GET
END_PROPERTY

METHOD PUBLIC ClearReference
VAR_INPUT
END_VAR
activeData REF= localData;
SetBaseDatatypeReference();
END_METHOD

METHOD PUBLIC Clone : I_Datatype
VAR
    pClone : POINTER TO _TcVnVector2_REAL;
END_VAR
pClone := __NEW(_TcVnVector2_REAL);
Clone := pClone^;
END_METHOD

METHOD FB_init : BOOL
VAR_INPUT
	bInitRetains : BOOL; // if TRUE, the retain variables are initialized (warm start / cold start)
	bInCopyCode : BOOL;  // if TRUE, the instance afterwards gets moved into the copy code (online change)
	//InitialValue : <type>; // if possible, not all values can be initialized
END_VAR
//localData := InitialValue; // if possible, not all values can be initialized
SetBaseDatatypeReference();
AddBaseDatatype(aliasBaseDatatype);
END_METHOD

PROPERTY PUBLIC Identifier : T_MAXSTRING
GET
Identifier := 'TcVnVector2_REAL';
END_GET
END_PROPERTY

METHOD PUBLIC MakeReferenceTo
VAR_INPUT
	ReferenceTarget : REFERENCE TO TcVnVector2_REAL;
END_VAR
activeData REF= ReferenceTarget;
SetBaseDatatypeReference();
END_METHOD

METHOD PROTECTED SetBaseDatatypeReference
VAR_INPUT
END_VAR
aliasBaseDatatype.MakeReferenceTo(activeData);
END_METHOD

PROPERTY PUBLIC Size : UDINT
GET
Size := SIZEOF(activeData);
END_GET
END_PROPERTY

METHOD TryMakeReferenceTo : BOOL
VAR_INPUT
	Target : I_Datatype;
END_VAR
VAR
	pTargetData : POINTER TO TcVnVector2_REAL;
END_VAR
IF NOT IsEquivalentTo(Target) THEN
	RETURN;
END_IF

pTargetData := Target.Address;
activeData REF= pTargetData^;
SetBaseDatatypeReference();
TryMakeReferenceTo := TRUE;
END_METHOD

PROPERTY PUBLIC Value : REFERENCE TO TcVnVector2_REAL
GET
Value REF= activeData;
END_GET
END_PROPERTY

END_FUNCTION_BLOCK

// ---- Datatypes/Arrays/_Array0to1OfREAL.TcPOU
{attribute 'linkalways'} 
{attribute 'no_explicit_call' := 'This FB is a CLASS and must be accessed using methods or properties'}
{attribute 'enable_dynamic_creation'}
FUNCTION_BLOCK _Array0to1OfREAL EXTENDS ArrayDatatypeBase_1D
VAR CONSTANT
	lBound : DINT := 0;
	uBound : DINT := 1;
END_VAR
VAR
	localData : ARRAY [lBound..uBound] OF REAL;
	activeData : REFERENCE TO ARRAY [lBound..uBound] OF REAL REF= localData;
	elements : ARRAY [lBound..uBound] OF _REAL(0.0);
	baseType : _REAL(0.0);
END_VAR

PROPERTY PUBLIC Address : PVOID
GET
Address := ADR(activeData);
END_GET
END_PROPERTY

PROPERTY PUBLIC BaseDatatype : I_Datatype
GET
BaseDatatype := baseType;
END_GET
END_PROPERTY

METHOD PUBLIC ClearReference
VAR_INPUT
END_VAR
activeData REF= localData;
SetElementReference();
END_METHOD

METHOD PUBLIC Clone : I_Datatype
VAR
    pClone : POINTER TO _Array0to1OfREAL;
END_VAR
pClone := __NEW(_Array0to1OfREAL());
pClone^.Value := Value;
Clone := pClone^;
END_METHOD

METHOD FB_init : BOOL
VAR_INPUT
	bInitRetains : BOOL; // if TRUE, the retain variables are initialized (warm start / cold start)
	bInCopyCode : BOOL;  // if TRUE, the instance afterwards gets moved into the copy code (online change)
END_VAR
SetElementReference();
END_METHOD

METHOD PUBLIC MakeReferenceTo
VAR_INPUT
	ReferenceTarget : REFERENCE TO ARRAY [lBound..uBound] OF REAL;
END_VAR
activeData REF= ReferenceTarget;
SetElementReference();
END_METHOD

METHOD PROTECTED OnSerializeArrayValues
VAR_INPUT
	Serializer : I_Serializer;
END_VAR
VAR
	i : DINT;
END_VAR
FOR i := lBound TO uBound DO
	elements[i].SerializeWith(Serializer);
END_FOR
END_METHOD

METHOD PROTECTED SetElementReference
VAR_INPUT
END_VAR
VAR
	i : DINT;
END_VAR
FOR i := lBound TO uBound DO
	elements[i].MakeReferenceTo(activeData[i]);
END_FOR
END_METHOD

PROPERTY PUBLIC Size : UDINT
GET
Size := SIZEOF(activeData);
END_GET
END_PROPERTY

METHOD PROTECTED TryDeserializeArrayValues : BOOL
VAR_INPUT
	Deserializer : I_Deserializer;
	Feedback : I_DeserializerFeedback;
END_VAR
VAR
	enumerator : I_DeserializerArrayForwardEnumerator;
	i : DINT;
END_VAR
enumerator := Deserializer.GetArrayEnumerator();
i := lBound;

WHILE enumerator.MoveNext() AND i <= uBound DO
	
	IF NOT elements[i].TryDeserializeFrom(enumerator.Current, Feedback) THEN
		EXIT;
	END_IF
	i := i + 1;

END_WHILE
enumerator.Dispose();
END_METHOD

METHOD PUBLIC TryGetElementAsDatatypeByIndex : BOOL
VAR_INPUT
	Index : DINT;
	Destination : REFERENCE TO I_Datatype;
END_VAR
IF Index < lbound OR Index > ubound THEN
	RETURN;
END_IF

Destination := elements[Index];
TryGetElementAsDatatypeByIndex := TRUE;
END_METHOD

METHOD PUBLIC TryGetLowerBound : BOOL
VAR_INPUT
	Dimention : UDINT;
	Destination : REFERENCE TO DINT;
END_VAR
IF Dimention = 1 THEN
	Destination := lBound;
	TryGetLowerBound := TRUE;
END_IF
END_METHOD

METHOD PUBLIC TryGetUpperBound : BOOL
VAR_INPUT
	Dimention : UDINT;
	Destination : REFERENCE TO DINT;
END_VAR
IF Dimention = 1 THEN
	Destination := uBound;
	TryGetUpperBound := TRUE;
END_IF
END_METHOD

METHOD TryMakeReferenceTo : BOOL
VAR_INPUT
	Target : I_Datatype;
END_VAR
VAR
	pTargetData : POINTER TO ARRAY [lBound..uBound] OF REAL;
END_VAR
IF NOT IsEquivalentTo(Target) THEN
	RETURN;
END_IF

pTargetData := Target.Address;
activeData REF= pTargetData^;
SetElementReference();
TryMakeReferenceTo := TRUE;
END_METHOD

PROPERTY PUBLIC Value : REFERENCE TO ARRAY [lBound..uBound] OF REAL;
GET
Value ref= activeData;
END_GET
END_PROPERTY

END_FUNCTION_BLOCK

// ---- Datatypes/Aliases/_TcVnArray4_LREAL.TcPOU
{attribute 'linkalways'} 
{attribute 'no_explicit_call' := 'This FB is a CLASS and must be accessed using methods or properties'}
{attribute 'enable_dynamic_creation'}
FUNCTION_BLOCK _TcVnArray4_LREAL EXTENDS AliasDatatypeBase
VAR
	localData : TcVnArray4_LREAL;
	activeData : REFERENCE TO TcVnArray4_LREAL REF= localData;
	aliasBaseDatatype : _Array0to3OfLREAL;
END_VAR

PROPERTY PUBLIC Address : PVOID
GET
Address := ADR(activeData);
END_GET
END_PROPERTY

METHOD PUBLIC ClearReference
VAR_INPUT
END_VAR
activeData REF= localData;
SetBaseDatatypeReference();
END_METHOD

METHOD PUBLIC Clone : I_Datatype
VAR
    pClone : POINTER TO _TcVnArray4_LREAL;
END_VAR
pClone := __NEW(_TcVnArray4_LREAL);
Clone := pClone^;
END_METHOD

METHOD FB_init : BOOL
VAR_INPUT
	bInitRetains : BOOL; // if TRUE, the retain variables are initialized (warm start / cold start)
	bInCopyCode : BOOL;  // if TRUE, the instance afterwards gets moved into the copy code (online change)
	//InitialValue : TcVnArray4_LREAL; // if possible, not all values can be initialized
END_VAR
//localData := InitialValue; // if possible, not all values can be initialized
SetBaseDatatypeReference();
AddBaseDatatype(aliasBaseDatatype);
END_METHOD

PROPERTY PUBLIC Identifier : T_MAXSTRING
GET
Identifier := 'TcVnArray4_LREAL';
END_GET
END_PROPERTY

METHOD PUBLIC MakeReferenceTo
VAR_INPUT
	ReferenceTarget : REFERENCE TO TcVnArray4_LREAL;
END_VAR
activeData REF= ReferenceTarget;
SetBaseDatatypeReference();
END_METHOD

METHOD PROTECTED SetBaseDatatypeReference
VAR_INPUT
END_VAR
aliasBaseDatatype.MakeReferenceTo(activeData);
END_METHOD

PROPERTY PUBLIC Size : UDINT
GET
Size := SIZEOF(activeData);
END_GET
END_PROPERTY

METHOD TryMakeReferenceTo : BOOL
VAR_INPUT
	Target : I_Datatype;
END_VAR
VAR
	pTargetData : POINTER TO TcVnArray4_LREAL;
END_VAR
IF NOT IsEquivalentTo(Target) THEN
	RETURN;
END_IF

pTargetData := Target.Address;
activeData REF= pTargetData^;
SetBaseDatatypeReference();
TryMakeReferenceTo := TRUE;
END_METHOD

PROPERTY PUBLIC Value : REFERENCE TO TcVnArray4_LREAL
GET
Value REF= activeData;
END_GET
END_PROPERTY

END_FUNCTION_BLOCK

// ---- Datatypes/Arrays/_Array0to3OfLREAL.TcPOU
{attribute 'linkalways'} 
{attribute 'no_explicit_call' := 'This FB is a CLASS and must be accessed using methods or properties'}
{attribute 'enable_dynamic_creation'}
FUNCTION_BLOCK _Array0to3OfLREAL EXTENDS ArrayDatatypeBase_1D
VAR CONSTANT
	lBound : DINT := 0;
	uBound : DINT := 3;
END_VAR
VAR
	localData : ARRAY [lBound..uBound] OF LREAL;
	activeData : REFERENCE TO ARRAY [lBound..uBound] OF LREAL REF= localData;
	elements : ARRAY [lBound..uBound] OF _LREAL(0.0);
	baseType : _LREAL(0.0);
END_VAR

PROPERTY PUBLIC Address : PVOID
GET
Address := ADR(activeData);
END_GET
END_PROPERTY

PROPERTY PUBLIC BaseDatatype : I_Datatype
GET
BaseDatatype := baseType;
END_GET
END_PROPERTY

METHOD PUBLIC ClearReference
VAR_INPUT
END_VAR
activeData REF= localData;
SetElementReference();
END_METHOD

METHOD PUBLIC Clone : I_Datatype
VAR
    pClone : POINTER TO _Array0to3OfLREAL;
END_VAR
pClone := __NEW(_Array0to3OfLREAL());
pClone^.Value := Value;
Clone := pClone^;
END_METHOD

METHOD FB_init : BOOL
VAR_INPUT
	bInitRetains : BOOL; // if TRUE, the retain variables are initialized (warm start / cold start)
	bInCopyCode : BOOL;  // if TRUE, the instance afterwards gets moved into the copy code (online change)
END_VAR
SetElementReference();
END_METHOD

METHOD PUBLIC MakeReferenceTo
VAR_INPUT
	ReferenceTarget : REFERENCE TO ARRAY [lBound..uBound] OF LREAL;
END_VAR
activeData REF= ReferenceTarget;
SetElementReference();
END_METHOD

METHOD PROTECTED OnSerializeArrayValues
VAR_INPUT
	Serializer : I_Serializer;
END_VAR
VAR
	i : DINT;
END_VAR
FOR i := lBound TO uBound DO
	elements[i].SerializeWith(Serializer);
END_FOR
END_METHOD

METHOD PROTECTED SetElementReference
VAR_INPUT
END_VAR
VAR
	i : DINT;
END_VAR
FOR i := lBound TO uBound DO
	elements[i].MakeReferenceTo(activeData[i]);
END_FOR
END_METHOD

PROPERTY PUBLIC Size : UDINT
GET
Size := SIZEOF(activeData);
END_GET
END_PROPERTY

METHOD PROTECTED TryDeserializeArrayValues : BOOL
VAR_INPUT
	Deserializer : I_Deserializer;
	Feedback : I_DeserializerFeedback;
END_VAR
VAR
	enumerator : I_DeserializerArrayForwardEnumerator;
	i : DINT;
END_VAR
enumerator := Deserializer.GetArrayEnumerator();
i := lBound;

WHILE enumerator.MoveNext() AND i <= uBound DO
	
	IF NOT elements[i].TryDeserializeFrom(enumerator.Current, Feedback) THEN
		EXIT;
	END_IF
	i := i + 1;

END_WHILE
enumerator.Dispose();
END_METHOD

METHOD PUBLIC TryGetElementAsDatatypeByIndex : BOOL
VAR_INPUT
	Index : DINT;
	Destination : REFERENCE TO I_Datatype;
END_VAR
IF Index < lbound OR Index > ubound THEN
	RETURN;
END_IF

Destination := elements[Index];
TryGetElementAsDatatypeByIndex := TRUE;
END_METHOD

METHOD PUBLIC TryGetLowerBound : BOOL
VAR_INPUT
	Dimention : UDINT;
	Destination : REFERENCE TO DINT;
END_VAR
IF Dimention = 1 THEN
	Destination := lBound;
	TryGetLowerBound := TRUE;
END_IF
END_METHOD

METHOD PUBLIC TryGetUpperBound : BOOL
VAR_INPUT
	Dimention : UDINT;
	Destination : REFERENCE TO DINT;
END_VAR
IF Dimention = 1 THEN
	Destination := uBound;
	TryGetUpperBound := TRUE;
END_IF
END_METHOD

METHOD TryMakeReferenceTo : BOOL
VAR_INPUT
	Target : I_Datatype;
END_VAR
VAR
	targetAsArray : I_ArrayDatatype;
	pTargetData : POINTER TO ARRAY [lBound..uBound] OF LREAL;
END_VAR
IF NOT Target.TryResolveAsArrayDatatype(targetAsArray) THEN
	RETURN;
END_IF

IF NOT (targetAsArray.Identifier = Identifier) THEN
	RETURN;
END_IF

pTargetData := Target.Address;
activeData REF= pTargetData^;
SetElementReference();
TryMakeReferenceTo := TRUE;
END_METHOD

PROPERTY PUBLIC Value : REFERENCE TO ARRAY [lBound..uBound] OF LREAL;
GET
Value ref= activeData;
END_GET
END_PROPERTY

END_FUNCTION_BLOCK

// ---- Datatypes/Aliases/_TcVnArray33_UDINT.TcPOU
{attribute 'linkalways'} 
{attribute 'no_explicit_call' := 'This FB is a CLASS and must be accessed using methods or properties'}
{attribute 'enable_dynamic_creation'}
FUNCTION_BLOCK _TcVnArray33_UDINT EXTENDS AliasDatatypeBase
VAR
	localData : TcVnArray33_UDINT;
	activeData : REFERENCE TO TcVnArray33_UDINT REF= localData;
	aliasBaseDatatype : _Array0to32OfUDINT;
END_VAR

PROPERTY PUBLIC Address : PVOID
GET
Address := ADR(activeData);
END_GET
END_PROPERTY

METHOD PUBLIC ClearReference
VAR_INPUT
END_VAR
activeData REF= localData;
SetBaseDatatypeReference();
END_METHOD

METHOD PUBLIC Clone : I_Datatype
VAR
    pClone : POINTER TO _TcVnArray33_UDINT;
END_VAR
pClone := __NEW(_TcVnArray33_UDINT);
Clone := pClone^;
END_METHOD

METHOD FB_init : BOOL
VAR_INPUT
	bInitRetains : BOOL; // if TRUE, the retain variables are initialized (warm start / cold start)
	bInCopyCode : BOOL;  // if TRUE, the instance afterwards gets moved into the copy code (online change)
	//InitialValue : TcVnArray33_UDINT; // if possible, not all values can be initialized
END_VAR
//localData := InitialValue; // if possible, not all values can be initialized
SetBaseDatatypeReference();
AddBaseDatatype(aliasBaseDatatype);
END_METHOD

PROPERTY PUBLIC Identifier : T_MAXSTRING
GET
Identifier := 'TcVnArray33_UDINT';
END_GET
END_PROPERTY

METHOD PUBLIC MakeReferenceTo
VAR_INPUT
	ReferenceTarget : REFERENCE TO TcVnArray33_UDINT;
END_VAR
activeData REF= ReferenceTarget;
SetBaseDatatypeReference();
END_METHOD

METHOD PROTECTED SetBaseDatatypeReference
VAR_INPUT
END_VAR
aliasBaseDatatype.MakeReferenceTo(activeData);
END_METHOD

PROPERTY PUBLIC Size : UDINT
GET
Size := SIZEOF(activeData);
END_GET
END_PROPERTY

METHOD TryMakeReferenceTo : BOOL
VAR_INPUT
	Target : I_Datatype;
END_VAR
VAR
	pTargetData : POINTER TO TcVnArray33_UDINT;
END_VAR
IF NOT IsEquivalentTo(Target) THEN
	RETURN;
END_IF

pTargetData := Target.Address;
activeData REF= pTargetData^;
SetBaseDatatypeReference();
TryMakeReferenceTo := TRUE;
END_METHOD

PROPERTY PUBLIC Value : REFERENCE TO TcVnArray33_UDINT
GET
Value REF= activeData;
END_GET
END_PROPERTY

END_FUNCTION_BLOCK

// ---- Datatypes/Arrays/_Array0to32OfUDINT.TcPOU
{attribute 'linkalways'} 
{attribute 'no_explicit_call' := 'This FB is a CLASS and must be accessed using methods or properties'}
{attribute 'enable_dynamic_creation'}
FUNCTION_BLOCK _Array0to32OfUDINT EXTENDS ArrayDatatypeBase_1D
VAR CONSTANT
	lBound : DINT := 0;
	uBound : DINT := 32;
END_VAR
VAR
	localData : ARRAY [lBound..uBound] OF UDINT;
	activeData : REFERENCE TO ARRAY [lBound..uBound] OF UDINT REF= localData;
	elements : ARRAY [lBound..uBound] OF _UDINT(0);
	baseType : _UDINT(0);
END_VAR

PROPERTY PUBLIC Address : PVOID
GET
Address := ADR(activeData);
END_GET
END_PROPERTY

PROPERTY PUBLIC BaseDatatype : I_Datatype
GET
BaseDatatype := baseType;
END_GET
END_PROPERTY

METHOD PUBLIC ClearReference
VAR_INPUT
END_VAR
activeData REF= localData;
SetElementReference();
END_METHOD

METHOD PUBLIC Clone : I_Datatype
VAR
    pClone : POINTER TO _Array0to32OfUDINT;
END_VAR
pClone := __NEW(_Array0to32OfUDINT());
pClone^.Value := Value;
Clone := pClone^;
END_METHOD

METHOD FB_init : BOOL
VAR_INPUT
	bInitRetains : BOOL; // if TRUE, the retain variables are initialized (warm start / cold start)
	bInCopyCode : BOOL;  // if TRUE, the instance afterwards gets moved into the copy code (online change)
END_VAR
SetElementReference();
END_METHOD

METHOD PUBLIC MakeReferenceTo
VAR_INPUT
	ReferenceTarget : REFERENCE TO ARRAY [lBound..uBound] OF UDINT;
END_VAR
activeData REF= ReferenceTarget;
SetElementReference();
END_METHOD

METHOD PROTECTED OnSerializeArrayValues
VAR_INPUT
	Serializer : I_Serializer;
END_VAR
VAR
	i : DINT;
END_VAR
FOR i := lBound TO uBound DO
	elements[i].SerializeWith(Serializer);
END_FOR
END_METHOD

METHOD PROTECTED SetElementReference
VAR_INPUT
END_VAR
VAR
	i : DINT;
END_VAR
FOR i := lBound TO uBound DO
	elements[i].MakeReferenceTo(activeData[i]);
END_FOR
END_METHOD

PROPERTY PUBLIC Size : UDINT
GET
Size := SIZEOF(activeData);
END_GET
END_PROPERTY

METHOD PROTECTED TryDeserializeArrayValues : BOOL
VAR_INPUT
	Deserializer : I_Deserializer;
	Feedback : I_DeserializerFeedback;
END_VAR
VAR
	enumerator : I_DeserializerArrayForwardEnumerator;
	i : DINT;
END_VAR
enumerator := Deserializer.GetArrayEnumerator();
i := lBound;

WHILE enumerator.MoveNext() AND i <= uBound DO
	
	IF NOT elements[i].TryDeserializeFrom(enumerator.Current, Feedback) THEN
		EXIT;
	END_IF
	i := i + 1;

END_WHILE
enumerator.Dispose();
END_METHOD

METHOD PUBLIC TryGetElementAsDatatypeByIndex : BOOL
VAR_INPUT
	Index : DINT;
	Destination : REFERENCE TO I_Datatype;
END_VAR
IF Index < lbound OR Index > ubound THEN
	RETURN;
END_IF

Destination := elements[Index];
TryGetElementAsDatatypeByIndex := TRUE;
END_METHOD

METHOD PUBLIC TryGetLowerBound : BOOL
VAR_INPUT
	Dimention : UDINT;
	Destination : REFERENCE TO DINT;
END_VAR
IF Dimention = 1 THEN
	Destination := lBound;
	TryGetLowerBound := TRUE;
END_IF
END_METHOD

METHOD PUBLIC TryGetUpperBound : BOOL
VAR_INPUT
	Dimention : UDINT;
	Destination : REFERENCE TO DINT;
END_VAR
IF Dimention = 1 THEN
	Destination := uBound;
	TryGetUpperBound := TRUE;
END_IF
END_METHOD

METHOD TryMakeReferenceTo : BOOL
VAR_INPUT
	Target : I_Datatype;
END_VAR
VAR
	pTargetData : POINTER TO ARRAY [lBound..uBound] OF UDINT;
END_VAR
IF NOT IsEquivalentTo(Target) THEN
	RETURN;
END_IF

pTargetData := Target.Address;
activeData REF= pTargetData^;
SetElementReference();
TryMakeReferenceTo := TRUE;
END_METHOD

PROPERTY PUBLIC Value : REFERENCE TO ARRAY [lBound..uBound] OF UDINT;
GET
Value ref= activeData;
END_GET
END_PROPERTY

END_FUNCTION_BLOCK

// ---- Datatypes/Aliases/_TcVnArray10_ITcVnImage.TcPOU
{attribute 'linkalways'} 
{attribute 'no_explicit_call' := 'This FB is a CLASS and must be accessed using methods or properties'}
{attribute 'enable_dynamic_creation'}
FUNCTION_BLOCK _TcVnArray10_ITcVnImage EXTENDS AliasDatatypeBase
VAR
	localData : TcVnArray10_ITcVnImage;
	activeData : REFERENCE TO TcVnArray10_ITcVnImage REF= localData;
	aliasBaseDatatype : _Array0to9OfITcVnImage;
END_VAR

PROPERTY PUBLIC Address : PVOID
GET
Address := ADR(activeData);
END_GET
END_PROPERTY

METHOD PUBLIC ClearReference
VAR_INPUT
END_VAR
activeData REF= localData;
SetBaseDatatypeReference();
END_METHOD

METHOD PUBLIC Clone : I_Datatype
VAR
    pClone : POINTER TO _TcVnArray10_ITcVnImage;
END_VAR
pClone := __NEW(_TcVnArray10_ITcVnImage);
Clone := pClone^;
END_METHOD

METHOD FB_init : BOOL
VAR_INPUT
	bInitRetains : BOOL; // if TRUE, the retain variables are initialized (warm start / cold start)
	bInCopyCode : BOOL;  // if TRUE, the instance afterwards gets moved into the copy code (online change)
	//InitialValue : TcVnArray10_ITcVnImage; // if possible, not all values can be initialized
END_VAR
//localData := InitialValue; // if possible, not all values can be initialized
SetBaseDatatypeReference();
AddBaseDatatype(aliasBaseDatatype);
END_METHOD

PROPERTY PUBLIC Identifier : T_MAXSTRING
GET
Identifier := 'TcVnArray10_ITcVnImage';
END_GET
END_PROPERTY

METHOD PUBLIC MakeReferenceTo
VAR_INPUT
	ReferenceTarget : REFERENCE TO TcVnArray10_ITcVnImage;
END_VAR
activeData REF= ReferenceTarget;
SetBaseDatatypeReference();
END_METHOD

METHOD PROTECTED SetBaseDatatypeReference
VAR_INPUT
END_VAR
aliasBaseDatatype.MakeReferenceTo(activeData);
END_METHOD

PROPERTY PUBLIC Size : UDINT
GET
Size := SIZEOF(activeData);
END_GET
END_PROPERTY

METHOD TryMakeReferenceTo : BOOL
VAR_INPUT
	Target : I_Datatype;
END_VAR
VAR
	pTargetData : POINTER TO TcVnArray10_ITcVnImage;
END_VAR
IF NOT IsEquivalentTo(Target) THEN
	RETURN;
END_IF

pTargetData := Target.Address;
activeData REF= pTargetData^;
SetBaseDatatypeReference();
TryMakeReferenceTo := TRUE;
END_METHOD

PROPERTY PUBLIC Value : REFERENCE TO TcVnArray10_ITcVnImage
GET
Value REF= activeData;
END_GET
END_PROPERTY

END_FUNCTION_BLOCK

// ---- Datatypes/Arrays/_Array0to9OfITcVnImage.TcPOU
{attribute 'linkalways'} 
{attribute 'no_explicit_call' := 'This FB is a CLASS and must be accessed using methods or properties'}
{attribute 'enable_dynamic_creation'}
FUNCTION_BLOCK _Array0to9OfITcVnImage EXTENDS ArrayDatatypeBase_1D
VAR CONSTANT
	lBound : DINT := 0;
	uBound : DINT := 9;
END_VAR
VAR
	localData : ARRAY [lBound..uBound] OF ITcVnImage;
	activeData : REFERENCE TO ARRAY [lBound..uBound] OF ITcVnImage REF= localData;
	elements : ARRAY [lBound..uBound] OF _ITcVnImage;
	baseType : _ITcVnImage;
END_VAR

PROPERTY PUBLIC Address : PVOID
GET
Address := ADR(activeData);
END_GET
END_PROPERTY

PROPERTY PUBLIC BaseDatatype : I_Datatype
GET
BaseDatatype := baseType;
END_GET
END_PROPERTY

METHOD PUBLIC ClearReference
VAR_INPUT
END_VAR
activeData REF= localData;
SetElementReference();
END_METHOD

METHOD PUBLIC Clone : I_Datatype
VAR
    pClone : POINTER TO _Array0to9OfITcVnImage;
END_VAR
pClone := __NEW(_Array0to9OfITcVnImage());
pClone^.Value := Value;
Clone := pClone^;
END_METHOD

METHOD FB_init : BOOL
VAR_INPUT
	bInitRetains : BOOL; // if TRUE, the retain variables are initialized (warm start / cold start)
	bInCopyCode : BOOL;  // if TRUE, the instance afterwards gets moved into the copy code (online change)
END_VAR
SetElementReference();
END_METHOD

METHOD PUBLIC MakeReferenceTo
VAR_INPUT
	ReferenceTarget : REFERENCE TO ARRAY [lBound..uBound] OF ITcVnImage;
END_VAR
activeData REF= ReferenceTarget;
SetElementReference();
END_METHOD

METHOD PROTECTED OnSerializeArrayValues
VAR_INPUT
	Serializer : I_Serializer;
END_VAR
VAR
	i : DINT;
END_VAR
FOR i := lBound TO uBound DO
	elements[i].SerializeWith(Serializer);
END_FOR
END_METHOD

METHOD PROTECTED SetElementReference
VAR_INPUT
END_VAR
VAR
	i : DINT;
END_VAR
FOR i := lBound TO uBound DO
	elements[i].MakeReferenceTo(activeData[i]);
END_FOR
END_METHOD

PROPERTY PUBLIC Size : UDINT
GET
Size := SIZEOF(activeData);
END_GET
END_PROPERTY

METHOD PROTECTED TryDeserializeArrayValues : BOOL
VAR_INPUT
	Deserializer : I_Deserializer;
	Feedback : I_DeserializerFeedback;
END_VAR
VAR
	enumerator : I_DeserializerArrayForwardEnumerator;
	i : DINT;
END_VAR
enumerator := Deserializer.GetArrayEnumerator();
i := lBound;

WHILE enumerator.MoveNext() AND i <= uBound DO
	
	IF NOT elements[i].TryDeserializeFrom(enumerator.Current, Feedback) THEN
		EXIT;
	END_IF
	i := i + 1;

END_WHILE
enumerator.Dispose();
END_METHOD

METHOD PUBLIC TryGetElementAsDatatypeByIndex : BOOL
VAR_INPUT
	Index : DINT;
	Destination : REFERENCE TO I_Datatype;
END_VAR
IF Index < lbound OR Index > ubound THEN
	RETURN;
END_IF

Destination := elements[Index];
TryGetElementAsDatatypeByIndex := TRUE;
END_METHOD

METHOD PUBLIC TryGetLowerBound : BOOL
VAR_INPUT
	Dimention : UDINT;
	Destination : REFERENCE TO DINT;
END_VAR
IF Dimention = 1 THEN
	Destination := lBound;
	TryGetLowerBound := TRUE;
END_IF
END_METHOD

METHOD PUBLIC TryGetUpperBound : BOOL
VAR_INPUT
	Dimention : UDINT;
	Destination : REFERENCE TO DINT;
END_VAR
IF Dimention = 1 THEN
	Destination := uBound;
	TryGetUpperBound := TRUE;
END_IF
END_METHOD

METHOD TryMakeReferenceTo : BOOL
VAR_INPUT
	Target : I_Datatype;
END_VAR
VAR
	targetAsArray : I_ArrayDatatype;
	pTargetData : POINTER TO ARRAY [lBound..uBound] OF ITcVnImage;
END_VAR
IF NOT Target.TryResolveAsArrayDatatype(targetAsArray) THEN
	RETURN;
END_IF

IF NOT (targetAsArray.Identifier = Identifier) THEN
	RETURN;
END_IF

pTargetData := Target.Address;
activeData REF= pTargetData^;
SetElementReference();
TryMakeReferenceTo := TRUE;
END_METHOD

PROPERTY PUBLIC Value : REFERENCE TO ARRAY [lBound..uBound] OF ITcVnImage;
GET
Value ref= activeData;
END_GET
END_PROPERTY

END_FUNCTION_BLOCK

// ---- Datatypes/Interfaces/_ITcVnImage.TcPOU
{attribute 'linkalways'} 
{attribute 'no_explicit_call' := 'This FB is a CLASS and must be accessed using methods or properties'}
{attribute 'enable_dynamic_creation'}
FUNCTION_BLOCK _ITcVnImage EXTENDS InterfaceDatatypeBase
VAR
	localData : ITcVnImage;
	activeData : REFERENCE TO ITcVnImage REF= localData;
END_VAR

PROPERTY PUBLIC Address : PVOID
GET
Address := ADR(activeData);
END_GET
END_PROPERTY

METHOD PUBLIC ClearReference
VAR_INPUT
END_VAR
activeData REF= localData;
END_METHOD

METHOD PUBLIC Clone : I_Datatype
VAR
    pClone : POINTER TO _ITcVnImage;
END_VAR
pClone := __NEW(_ITcVnImage);
Clone := pClone^;
END_METHOD

METHOD FB_exit : BOOL
VAR_INPUT
	bInCopyCode : BOOL; // if TRUE, the exit method is called for exiting an instance that is copied afterwards (online change).
END_VAR
IF bInCopyCode THEN
	RETURN;
END_IF

TryTcReleaseLocal();
END_METHOD

METHOD PUBLIC HasChannelCount : BOOL
VAR_INPUT
	ChannelCount : BYTE;
END_VAR
VAR
    pixelFormat : TcVnPixelFormat;
END_VAR
IF NOT TryGetPixelFormat(pixelFormat) THEN
    RETURN;
END_IF

IF NOT (pixelFormat.nChannels = ChannelCount) THEN
    RETURN;
END_IF

HasChannelCount := TRUE;
END_METHOD

PROPERTY PUBLIC Identifier : T_MAXSTRING
GET
Identifier := 'ITcVnImage';
END_GET
END_PROPERTY

METHOD PUBLIC IsPixelDepth : BOOL
VAR_INPUT
	PixelDepth : UINT;
END_VAR
VAR
    pixelFormat : TcVnPixelFormat;
END_VAR
IF NOT TryGetPixelFormat(pixelFormat) THEN
    RETURN;
END_IF

IF NOT (pixelFormat.nElementSize = PixelDepth) THEN
    RETURN;
END_IF

IsPixelDepth := TRUE;
END_METHOD

PROPERTY PUBLIC IsValid : BOOL
GET
IsValid := activeData <> 0;
END_GET
END_PROPERTY

METHOD PUBLIC MakeReferenceTo
VAR_INPUT
	ReferenceTarget : REFERENCE TO ITcVnImage;
END_VAR
activeData REF= ReferenceTarget;
END_METHOD

METHOD PUBLIC SerializeWith
VAR_INPUT
	Serializer : I_Serializer;
END_VAR
VAR
	result: HRESULT;
	exportImageSize: ULINT;
	buffer : POINTER TO BYTE;
	imageInfo : _TcVnImageInfo;
END_VAR
IF NOT (activeData <> 0) THEN
	// no image available, so drop out.. need to add serialization?
	Serializer.AddNull();
	RETURN;
END_IF

result := F_VN_ExportImageSize(ipImage:=activeData, nBufferSize:=exportImageSize, hrPrev:=result);

IF FAILED(result) THEN
	// export to bmp size failed, so drop out.. need to add serialization?
	Serializer.AddNull();
	RETURN;
END_IF

IF exportImageSize > DatatypeLimits.UDINT_MAX_VALUE THEN
	// export is too big for __NEW, so drop out..
	Serializer.AddNull();
	RETURN;
END_IF

IF exportImageSize <= 0 THEN
	// export is zero size, so drop out.. 
	Serializer.AddNull();
	RETURN;
END_IF
	
buffer := __NEW(BYTE,ULINT_TO_UDINT(exportImageSize));
result := F_VN_ExportImage(ipImage:=activeData, pBuffer:=buffer, nBufferSize:=exportImageSize, hrPrev:=result);

IF FAILED(result) THEN
	// export to bmp failed, so drop out.. 
	Serializer.AddNull();
	__DELETE(buffer);
	RETURN;
END_IF

activeData.GetImageInfo(imageInfo.value);

Serializer.StartObject();
Serializer.AddKeyObject('imageInfo',imageInfo);
Serializer.AddKey('imageData');
Serializer.AddBase64(buffer,ULINT_TO_DINT(exportImageSize));
Serializer.EndObject();

__DELETE(buffer);
END_METHOD

PROPERTY PUBLIC Size : UDINT
GET
Size := SIZEOF(activeData);
END_GET
END_PROPERTY

METHOD TryDeserializeFrom : BOOL
VAR_INPUT
	Deserializer : I_Deserializer;
	Feedback : I_DeserializerFeedback;
END_VAR
VAR
	imageInfo : _TcVnImageInfo;
	imageSizeInBytes : UDINT;
	buffer : POINTER TO BYTE;
	hr : HRESULT;
	elementType : ETcVnElementType;
END_VAR
IF NOT Deserializer.TryDeserializeKeyToObject('imageInfo', imageInfo, Feedback) THEN
	RETURN;
END_IF

imageSizeInBytes := ULINT_TO_UDINT(imageInfo.nImageSize.Value);

IF imageSizeInBytes = 0 THEN
	TryDeserializeFrom := TRUE;
	RETURN;
END_IF

buffer := __NEW(BYTE, imageSizeInBytes);

IF NOT Deserializer.TryGetKeyBase64('imageData', buffer, imageSizeInBytes, Feedback) THEN
	__DELETE(buffer);
	RETURN;
END_IF

TryGetElementTypeFromInfo(imageInfo.Value, elementType);

hr := F_VN_CreateImageFromArray(
	pData := buffer,
	ipImage := activeData,
	nWidth := imageInfo.nWidth.Value,
	nHeight :=  imageInfo.nHeight.Value,
	ePixelType := elementType,
	nChannelNum := imageInfo.stPixelFormat.nChannels.Value, 
	hrPrev := hr);

__DELETE(buffer);

TryDeserializeFrom := TRUE;
END_METHOD

METHOD PRIVATE TryGetElementTypeFromInfo : BOOL;
VAR_INPUT
	ImageInfo : TcVnImageInfo;
	Destination : REFERENCE TO ETcVnElementType;
END_VAR
CASE ImageInfo.stPixelFormat.nElementSize OF
	
	8 : // 8bit
	
		IF ImageInfo.stPixelFormat.bSigned THEN
			Destination := ETcVnElementType.TCVN_ET_SINT;
		ELSE	
			Destination := ETcVnElementType.TCVN_ET_USINT;
		END_IF
		TryGetElementTypeFromInfo := TRUE;
	
	16 : // 16bit
	
		IF ImageInfo.stPixelFormat.bSigned THEN
			Destination := ETcVnElementType.TCVN_ET_INT;
		ELSE	
			Destination := ETcVnElementType.TCVN_ET_UINT;
		END_IF
		TryGetElementTypeFromInfo := TRUE;
	
	32 : // 32bit
	
		IF ImageInfo.stPixelFormat.bSigned AND NOT ImageInfo.stPixelFormat.bFloat THEN
			Destination := ETcVnElementType.TCVN_ET_DINT;
			TryGetElementTypeFromInfo := TRUE;
		END_IF
		
		IF ImageInfo.stPixelFormat.bFloat THEN
			Destination := ETcVnElementType.TCVN_ET_REAL;
			TryGetElementTypeFromInfo := TRUE;
		END_IF
		
	64 : // 64bit
	
		IF ImageInfo.stPixelFormat.bFloat THEN
			Destination := ETcVnElementType.TCVN_ET_LREAL;
			TryGetElementTypeFromInfo := TRUE;
		END_IF
		
ELSE
	
	RETURN;

END_CASE
END_METHOD

METHOD PUBLIC TryGetHeight : BOOL
VAR_INPUT
	Destination : REFERENCE TO UDINT;
END_VAR
IF NOT IsValid THEN
	RETURN;
END_IF

TryGetHeight := SUCCEEDED(activeData.GetHeight(Destination));
END_METHOD

METHOD PUBLIC TryGetImageData : BOOL
VAR_INPUT
	Destination : POINTER TO ITcVnData;
END_VAR
IF NOT IsValid THEN
	RETURN;
END_IF

TryGetImageData := SUCCEEDED(activeData.GetImageData(Destination));
END_METHOD

METHOD PUBLIC TryGetImageInfo : BOOL
VAR_INPUT
	Destination : REFERENCE TO  TcVnImageInfo;
END_VAR
IF NOT IsValid THEN
	RETURN;
END_IF

TryGetImageInfo := SUCCEEDED(activeData.GetImageInfo(Destination));
END_METHOD

METHOD PUBLIC TryGetImageSize : BOOL
VAR_INPUT
	Destination : REFERENCE TO ULINT;
END_VAR
IF NOT IsValid THEN
	RETURN;
END_IF

TryGetImageSize := SUCCEEDED(activeData.GetImageSize(Destination));
END_METHOD

METHOD PUBLIC TryGetPixelFormat : BOOL
VAR_INPUT
	Destination : REFERENCE TO  TcVnPixelFormat;
END_VAR
IF NOT IsValid THEN
	RETURN;
END_IF

TryGetPixelFormat := SUCCEEDED(activeData.GetPixelFormat(Destination));
END_METHOD

METHOD PUBLIC TryGetRowPointer : BOOL
VAR_INPUT
	RowIndex : UDINT;
	Destination : POINTER TO PVOID;
END_VAR
IF NOT IsValid THEN
	RETURN;
END_IF

TryGetRowPointer := SUCCEEDED(activeData.GetRowPointer(RowIndex, Destination));
END_METHOD

METHOD PUBLIC TryGetWidth : BOOL
VAR_INPUT
	Destination : REFERENCE TO UDINT;
END_VAR
IF NOT IsValid THEN
	RETURN;
END_IF

TryGetWidth := SUCCEEDED(activeData.GetWidth(Destination));
END_METHOD

METHOD PUBLIC TryGetXPadding : BOOL
VAR_INPUT
	Destination : REFERENCE TO UINT;
END_VAR
IF NOT IsValid THEN
	RETURN;
END_IF

TryGetXPadding := SUCCEEDED(activeData.GetXPadding(Destination));
END_METHOD

METHOD PUBLIC TryGetYPadding : BOOL
VAR_INPUT
	Destination : REFERENCE TO UINT;
END_VAR
IF NOT IsValid THEN
	RETURN;
END_IF

TryGetYPadding := SUCCEEDED(activeData.GetYPadding(Destination));
END_METHOD

METHOD TryMakeReferenceTo : BOOL
VAR_INPUT
	Target : I_Datatype;
END_VAR
VAR
	pTargetData : POINTER TO ITcVnImage;
END_VAR
IF NOT IsEquivalentTo(Target) THEN
	RETURN;
END_IF

pTargetData := Target.Address;
activeData REF= pTargetData^;
TryMakeReferenceTo := TRUE;
END_METHOD

METHOD PUBLIC TryReleaseRowPointer : BOOL
VAR_INPUT
	ppRow : POINTER TO PVOID;
END_VAR
IF NOT IsValid THEN
	RETURN;
END_IF

TryReleaseRowPointer := SUCCEEDED(activeData.ReleaseRowPointer(ppRow));
END_METHOD

METHOD PUBLIC TryTcAddRef : BOOL
VAR_INPUT
END_VAR
IF activeData = 0 THEN
	RETURN;
END_IF

IF activeData.TcAddRef() = 0 THEN
	activeData := 0;
END_IF

TryTcAddRef := TRUE;
END_METHOD

METHOD PUBLIC TryTcRelease : BOOL
VAR_INPUT
END_VAR
IF activeData = 0 THEN
	RETURN;
END_IF

IF activeData.TcRelease() = 0 THEN
	activeData := 0;
END_IF

TryTcRelease := TRUE;
END_METHOD

METHOD PUBLIC TryTcReleaseLocal : BOOL
VAR_INPUT
END_VAR
IF localData = 0 THEN
	RETURN;
END_IF

IF localData.TcRelease() = 0 THEN
	localData := 0;
END_IF

TryTcReleaseLocal := TRUE;
END_METHOD

PROPERTY PUBLIC Value : REFERENCE TO ITcVnImage
GET
Value REF= activeData;
END_GET
END_PROPERTY

END_FUNCTION_BLOCK

// ---- Datatypes/Structs/_TcVnImageInfo.TcPOU
{attribute 'linkalways'} 
{attribute 'no_explicit_call' := 'This FB is a CLASS and must be accessed using methods or properties'}
{attribute 'enable_dynamic_creation'}
FUNCTION_BLOCK _TcVnImageInfo EXTENDS StructuredDatatypeBase
VAR
	localData : TcVnImageInfo;
	activeData : REFERENCE TO TcVnImageInfo REF= localData;
	_nImageSize : _ULINT(localData.nImageSize);
	_nWidth : _UDINT(localData.nWidth);
	_nHeight : _UDINT(localData.nHeight);
	_nXPadding : _UINT(localData.nXPadding);
	_nYPadding : _UINT(localData.nYPadding);
	_stPixelFormat : _TcVnPixelFormat();
END_VAR

PROPERTY PUBLIC Address : PVOID
GET
Address := ADR(activeData);
END_GET
END_PROPERTY

METHOD PUBLIC ClearReference
VAR_INPUT
END_VAR
activeData REF= localData;
SetMemberReference();
END_METHOD

METHOD PUBLIC Clone : I_Datatype
VAR
    pClone : POINTER TO _TcVnImageInfo;
END_VAR
pClone := __NEW(_TcVnImageInfo());
pClone^.Value := Value;
Clone := pClone^;
END_METHOD

METHOD FB_init : BOOL
VAR_INPUT
	bInitRetains : BOOL; // if TRUE, the retain variables are initialized (warm start / cold start)
	bInCopyCode : BOOL;  // if TRUE, the instance afterwards gets moved into the copy code (online change)
END_VAR
SetMemberReference();
AddMember('nImageSize',_nImageSize);
AddMember('nWidth',_nWidth);
AddMember('nHeight',_nHeight);
AddMember('nXPadding',_nXPadding);
AddMember('nYPadding',_nYPadding);
AddMember('stPixelFormat',_stPixelFormat);
END_METHOD

PROPERTY PUBLIC Identifier : T_MAXSTRING
GET
Identifier := 'TcVnImageInfo';
END_GET
END_PROPERTY

METHOD PUBLIC MakeReferenceTo
VAR_INPUT
	ReferenceTarget : REFERENCE TO TcVnImageInfo;
END_VAR
activeData REF= ReferenceTarget;
SetMemberReference();
END_METHOD

PROPERTY PUBLIC nHeight : Reference to _UDINT
GET
nHeight REF= _nHeight;
END_GET
END_PROPERTY

PROPERTY PUBLIC nImageSize : Reference to _ULINT
GET
nImageSize REF= _nImageSize;
END_GET
END_PROPERTY

PROPERTY PUBLIC nWidth : Reference to _UDINT
GET
nWidth REF= _nWidth;
END_GET
END_PROPERTY

PROPERTY PUBLIC nXPadding : Reference to _UINT
GET
nXPadding REF= _nXPadding;
END_GET
END_PROPERTY

PROPERTY PUBLIC nYPadding : Reference to _UINT
GET
nYPadding REF= _nYPadding;
END_GET
END_PROPERTY

METHOD PROTECTED SetMemberReference
VAR_INPUT
END_VAR
_nImageSize.MakeReferenceTo(activeData.nImageSize);
_nWidth.MakeReferenceTo(activeData.nWidth);
_nHeight.MakeReferenceTo(activeData.nHeight);
_nXPadding.MakeReferenceTo(activeData.nXPadding);
_nYPadding.MakeReferenceTo(activeData.nYPadding);
_stPixelFormat.MakeReferenceTo(activeData.stPixelFormat);
END_METHOD

PROPERTY PUBLIC Size : UDINT
GET
Size := SIZEOF(activeData);
END_GET
END_PROPERTY

PROPERTY PUBLIC stPixelFormat : Reference to _TcVnPixelFormat
GET
stPixelFormat REF= _stPixelFormat;
END_GET
END_PROPERTY

METHOD TryMakeReferenceTo : BOOL
VAR_INPUT
	Target : I_Datatype;
END_VAR
VAR
	pTargetData : POINTER TO TcVnImageInfo;
END_VAR
IF NOT IsEquivalentTo(Target) THEN
	RETURN;
END_IF

pTargetData := Target.Address;
activeData REF= pTargetData^;
SetMemberReference();
TryMakeReferenceTo := TRUE;
END_METHOD

PROPERTY PUBLIC Value : reference to TcVnImageInfo
GET
Value ref= activeData;
END_GET
END_PROPERTY

END_FUNCTION_BLOCK

// ---- Datatypes/Structs/_TcVnPixelFormat.TcPOU
{attribute 'linkalways'} 
{attribute 'no_explicit_call' := 'This FB is a CLASS and must be accessed using methods or properties'}
{attribute 'enable_dynamic_creation'}
FUNCTION_BLOCK _TcVnPixelFormat EXTENDS StructuredDatatypeBase
VAR
	localData : TcVnPixelFormat;
	activeData : REFERENCE TO TcVnPixelFormat REF= localData;

	_bSupported : _BIT();
	_bSigned : _BIT();
	_bPlanar : _BIT();
	_bFloat : _BIT();
	_nChannels : _BYTE(localData.nChannels);
	_ePixelEncoding : _ETcVnPixelEncoding(localData.ePixelEncoding);
	_ePixelPackMode : _ETcVnPixelPackMode(localData.ePixelPackMode);
	_nElementSize : _UINT(localData.nElementSize);
	_nTotalSize : _UINT(localData.nTotalSize);
END_VAR

PROPERTY PUBLIC Address : PVOID
GET
Address := ADR(activeData);
END_GET
END_PROPERTY

PROPERTY PUBLIC bFloat : Reference to _BIT
GET
bFloat REF= _bFloat;
END_GET
END_PROPERTY

PROPERTY PUBLIC bPlanar : Reference to _BIT
GET
bPlanar REF= _bPlanar;
END_GET
END_PROPERTY

PROPERTY PUBLIC bSigned : Reference to _BIT
GET
bSigned REF= _bSigned;
END_GET
END_PROPERTY

PROPERTY PUBLIC bSupported : Reference to _BIT
GET
bSupported REF= _bSupported;
END_GET
END_PROPERTY

METHOD PUBLIC ClearReference
VAR_INPUT
END_VAR
activeData REF= localData;
SetMemberReference();
END_METHOD

METHOD PUBLIC Clone : I_Datatype
VAR
    pClone : POINTER TO _TcVnPixelFormat;
END_VAR
pClone := __NEW(_TcVnPixelFormat());
pClone^.Value := Value;
Clone := pClone^;
END_METHOD

PROPERTY PUBLIC ePixelEncoding : Reference to _ETcVnPixelEncoding
GET
ePixelEncoding REF= _ePixelEncoding;
END_GET
END_PROPERTY

PROPERTY PUBLIC ePixelPackMode : Reference to _ETcVnPixelPackMode
GET
ePixelPackMode REF= _ePixelPackMode;
END_GET
END_PROPERTY

METHOD FB_init : BOOL
VAR_INPUT
	bInitRetains : BOOL; // if TRUE, the retain variables are initialized (warm start / cold start)
	bInCopyCode : BOOL;  // if TRUE, the instance afterwards gets moved into the copy code (online change)
END_VAR
SetMemberReference();
AddMember('bSupported',_bSupported);
AddMember('bSigned',_bSigned);
AddMember('bPlanar',_bPlanar);
AddMember('bFloat',_bFloat);
AddMember('nChannels',_nChannels);
AddMember('ePixelEncoding',_ePixelEncoding);
AddMember('ePixelPackMode',_ePixelPackMode);
AddMember('nElementSize',_nElementSize);
AddMember('nTotalSize',_nTotalSize);
END_METHOD

PROPERTY PUBLIC Identifier : T_MAXSTRING
GET
Identifier := 'TcVnPixelFormat';
END_GET
END_PROPERTY

METHOD PUBLIC MakeReferenceTo
VAR_INPUT
	ReferenceTarget : REFERENCE TO TcVnPixelFormat;
END_VAR
activeData REF= ReferenceTarget;
SetMemberReference();
END_METHOD

PROPERTY PUBLIC nChannels : Reference to _BYTE
GET
nChannels REF= _nChannels;
END_GET
END_PROPERTY

PROPERTY PUBLIC nElementSize : Reference to _UINT
GET
nElementSize REF= _nElementSize;
END_GET
END_PROPERTY

PROPERTY PUBLIC nTotalSize : Reference to _UINT
GET
nTotalSize REF= _nTotalSize;
END_GET
END_PROPERTY

METHOD PROTECTED SetMemberReference
VAR_STAT
	// this variable is used for BITADR as this function failes if used on a local variable.
	structure : TcVnPixelFormat;
END_VAR
_bSupported.MakeReferenceTo(THIS^, GetByteOffset(localData, localData.bSupported), BITADR(structure.bSupported));
_bSigned.MakeReferenceTo(THIS^, GetByteOffset(localData, localData.bSigned), BITADR(structure.bSigned));
_bPlanar.MakeReferenceTo(THIS^, GetByteOffset(localData, localData.bPlanar), BITADR(structure.bPlanar));
_bFloat.MakeReferenceTo(THIS^, GetByteOffset(localData, localData.bFloat), BITADR(structure.bFloat));
_nChannels.MakeReferenceTo(activeData.nChannels);
_ePixelEncoding.MakeReferenceTo(activeData.ePixelEncoding);
_ePixelPackMode.MakeReferenceTo(activeData.ePixelPackMode);
_nElementSize.MakeReferenceTo(activeData.nElementSize);
_nTotalSize.MakeReferenceTo(activeData.nTotalSize);
END_METHOD

PROPERTY PUBLIC Size : UDINT
GET
Size := SIZEOF(activeData);
END_GET
END_PROPERTY

METHOD TryMakeReferenceTo : BOOL
VAR_INPUT
	Target : I_Datatype;
END_VAR
VAR
	pTargetData : POINTER TO TcVnPixelFormat;
END_VAR
IF NOT IsEquivalentTo(Target) THEN
	RETURN;
END_IF

pTargetData := Target.Address;
activeData REF= pTargetData^;
SetMemberReference();
TryMakeReferenceTo := TRUE;
END_METHOD

PROPERTY PUBLIC Value : reference to TcVnPixelFormat
GET
Value REF= activeData;
END_GET
END_PROPERTY

END_FUNCTION_BLOCK

// ---- Datatypes/Enums/_ETcVnPixelEncoding.TcPOU
{attribute 'linkalways'} 
{attribute 'no_explicit_call' := 'This FB is a CLASS and must be accessed using methods or properties'}
{attribute 'enable_dynamic_creation'}
FUNCTION_BLOCK _ETcVnPixelEncoding EXTENDS EnumDatatypeBase
VAR
	localData : ETcVnPixelEncoding;
	activeData : REFERENCE TO ETcVnPixelEncoding;
	enumBaseDatatype : _BYTE(localData);
END_VAR

METHOD PRIVATE AddLocalEnumeration
VAR_INPUT
	Enumeration : T_MAXSTRING;
	Value : ETcVnPixelEncoding;
END_VAR
AddEnumeration(Enumeration, Value);
END_METHOD

PROPERTY PUBLIC Address : PVOID
GET
Address := ADR(activeData);
END_GET
END_PROPERTY

METHOD PUBLIC ClearReference
VAR_INPUT
END_VAR
activeData REF= localData;
SetBaseDatatypeReference();
END_METHOD

METHOD PUBLIC Clone : I_Datatype
VAR
    pClone : POINTER TO _ETcVnPixelEncoding;
END_VAR
pClone := __NEW(_ETcVnPixelEncoding(InitialValue := Value));
Clone := pClone^;
END_METHOD

METHOD FB_init : BOOL
VAR_INPUT
	bInitRetains : BOOL; // if TRUE, the retain variables are initialized (warm start / cold start)
	bInCopyCode : BOOL;  // if TRUE, the instance afterwards gets moved into the copy code (online change)
	InitialValue : ETcVnPixelEncoding;
END_VAR
localData := InitialValue;
AddBaseDatatype(enumBaseDatatype);
ClearReference();

AddLocalEnumeration('TCVN_PE_NONE', ETcVnPixelEncoding.TCVN_PE_NONE);
AddLocalEnumeration('TCVN_PE_BAYER_GR', ETcVnPixelEncoding.TCVN_PE_BAYER_GR);
AddLocalEnumeration('TCVN_PE_BAYER_RG', ETcVnPixelEncoding.TCVN_PE_BAYER_RG);
AddLocalEnumeration('TCVN_PE_BAYER_GB', ETcVnPixelEncoding.TCVN_PE_BAYER_GB);
AddLocalEnumeration('TCVN_PE_BAYER_BG', ETcVnPixelEncoding.TCVN_PE_BAYER_BG);
AddLocalEnumeration('TCVN_PE_YUV_411_UYYVYY', ETcVnPixelEncoding.TCVN_PE_YUV_411_UYYVYY);
AddLocalEnumeration('TCVN_PE_YUV_422_UYVY', ETcVnPixelEncoding.TCVN_PE_YUV_422_UYVY);
AddLocalEnumeration('TCVN_PE_YUV_422_YUYV', ETcVnPixelEncoding.TCVN_PE_YUV_422_YUYV);
AddLocalEnumeration('TCVN_PE_YCBCR_411_CBYYCRYY', ETcVnPixelEncoding.TCVN_PE_YCBCR_411_CBYYCRYY);
AddLocalEnumeration('TCVN_PE_YCBCR_422_CBYCRY', ETcVnPixelEncoding.TCVN_PE_YCBCR_422_CBYCRY);
AddLocalEnumeration('TCVN_PE_YCBCR_422_YCBYCR', ETcVnPixelEncoding.TCVN_PE_YCBCR_422_YCBYCR);
END_METHOD

PROPERTY PUBLIC Identifier : T_MAXSTRING
GET
Identifier := 'ETcVnPixelEncoding';
END_GET
END_PROPERTY

METHOD IsEnumeratorValueEqual : BOOL
VAR_INPUT
	Enumerator : I_KeyValueForwardEnumerator;
END_VAR
VAR
	storedValue : ETcVnPixelEncoding;
END_VAR
IF NOT Enumerator.TryGet(storedValue) THEN
	RETURN;
END_IF

IsEnumeratorValueEqual := storedValue = activeData;
END_METHOD

METHOD PUBLIC MakeReferenceTo
VAR_INPUT
	ReferenceTarget : REFERENCE TO ETcVnPixelEncoding;
END_VAR
activeData REF= ReferenceTarget;
SetBaseDatatypeReference();
END_METHOD

METHOD PROTECTED SetBaseDatatypeReference
VAR_INPUT
END_VAR
enumBaseDatatype.MakeReferenceTo(activeData);
END_METHOD

PROPERTY PUBLIC Size : UDINT
GET
Size := SIZEOF(activeData);
END_GET
END_PROPERTY

METHOD TryMakeReferenceTo : BOOL
VAR_INPUT
	Target : I_Datatype;
END_VAR
VAR
	pTargetData : POINTER TO ETcVnPixelEncoding;
END_VAR
IF NOT IsEquivalentTo(Target) THEN
	RETURN;
END_IF

pTargetData := Target.Address;
activeData REF= pTargetData^;
SetBaseDatatypeReference();
TryMakeReferenceTo := TRUE;
END_METHOD

PROPERTY PUBLIC Value : ETcVnPixelEncoding
GET
Value := activeData;
END_GET
SET
activeData := Value;
END_SET
END_PROPERTY

END_FUNCTION_BLOCK

// ---- Datatypes/Enums/_ETcVnPixelPackMode.TcPOU
{attribute 'linkalways'} 
{attribute 'no_explicit_call' := 'This FB is a CLASS and must be accessed using methods or properties'}
{attribute 'enable_dynamic_creation'}
FUNCTION_BLOCK _ETcVnPixelPackMode EXTENDS EnumDatatypeBase
VAR
	localData : ETcVnPixelPackMode;
	activeData : REFERENCE TO ETcVnPixelPackMode;
	enumBaseDatatype : _BYTE(localData);
END_VAR

METHOD PRIVATE AddLocalEnumeration
VAR_INPUT
	Enumeration : T_MAXSTRING;
	Value : ETcVnPixelPackMode;
END_VAR
AddEnumeration(Enumeration, Value);
END_METHOD

PROPERTY PUBLIC Address : PVOID
GET
Address := ADR(activeData);
END_GET
END_PROPERTY

METHOD PUBLIC ClearReference
VAR_INPUT
END_VAR
activeData REF= localData;
SetBaseDatatypeReference();
END_METHOD

METHOD PUBLIC Clone : I_Datatype
VAR
    pClone : POINTER TO _ETcVnPixelPackMode;
END_VAR
pClone := __NEW(_ETcVnPixelPackMode(InitialValue := Value));
Clone := pClone^;
END_METHOD

METHOD FB_init : BOOL
VAR_INPUT
	bInitRetains : BOOL; // if TRUE, the retain variables are initialized (warm start / cold start)
	bInCopyCode : BOOL;  // if TRUE, the instance afterwards gets moved into the copy code (online change)
	InitialValue : ETcVnPixelPackMode;
END_VAR
localData := InitialValue;
AddBaseDatatype(enumBaseDatatype);
ClearReference();

AddLocalEnumeration('TCVN_PPM_NONE', ETcVnPixelPackMode.TCVN_PPM_NONE);
AddLocalEnumeration('TCVN_PPM_MONO1P', ETcVnPixelPackMode.TCVN_PPM_MONO1P);
AddLocalEnumeration('TCVN_PPM_MONO2P', ETcVnPixelPackMode.TCVN_PPM_MONO2P);
AddLocalEnumeration('TCVN_PPM_MONO4P', ETcVnPixelPackMode.TCVN_PPM_MONO4P);
AddLocalEnumeration('TCVN_PPM_MONO10PACKED', ETcVnPixelPackMode.TCVN_PPM_MONO10PACKED);
AddLocalEnumeration('TCVN_PPM_MONO12PACKED', ETcVnPixelPackMode.TCVN_PPM_MONO12PACKED);
AddLocalEnumeration('TCVN_PPM_RGB10V1PACKED', ETcVnPixelPackMode.TCVN_PPM_RGB10V1PACKED);
AddLocalEnumeration('TCVN_PPM_RGB10P32', ETcVnPixelPackMode.TCVN_PPM_RGB10P32);
AddLocalEnumeration('TCVN_PPM_RGB12V1PACKED', ETcVnPixelPackMode.TCVN_PPM_RGB12V1PACKED);
AddLocalEnumeration('TCVN_PPM_RGB565P', ETcVnPixelPackMode.TCVN_PPM_RGB565P);
AddLocalEnumeration('TCVN_PPM_BGR565P', ETcVnPixelPackMode.TCVN_PPM_BGR565P);
AddLocalEnumeration('TCVN_PPM_MONO10P', ETcVnPixelPackMode.TCVN_PPM_MONO10P);
AddLocalEnumeration('TCVN_PPM_MONO12P', ETcVnPixelPackMode.TCVN_PPM_MONO12P);
END_METHOD

PROPERTY PUBLIC Identifier : T_MAXSTRING
GET
Identifier := 'ETcVnPixelPackMode';
END_GET
END_PROPERTY

METHOD IsEnumeratorValueEqual : BOOL
VAR_INPUT
	Enumerator : I_KeyValueForwardEnumerator;
END_VAR
VAR
	storedValue : ETcVnPixelPackMode;
END_VAR
IF NOT Enumerator.TryGet(storedValue) THEN
	RETURN;
END_IF

IsEnumeratorValueEqual := storedValue = activeData;
END_METHOD

METHOD PUBLIC MakeReferenceTo
VAR_INPUT
	ReferenceTarget : REFERENCE TO ETcVnPixelPackMode;
END_VAR
activeData REF= ReferenceTarget;
SetBaseDatatypeReference();
END_METHOD

METHOD PROTECTED SetBaseDatatypeReference
VAR_INPUT
END_VAR
enumBaseDatatype.MakeReferenceTo(activeData);
END_METHOD

PROPERTY PUBLIC Size : UDINT
GET
Size := SIZEOF(activeData);
END_GET
END_PROPERTY

METHOD TryMakeReferenceTo : BOOL
VAR_INPUT
	Target : I_Datatype;
END_VAR
VAR
	pTargetData : POINTER TO ETcVnPixelPackMode;
END_VAR
IF NOT IsEquivalentTo(Target) THEN
	RETURN;
END_IF

pTargetData := Target.Address;
activeData REF= pTargetData^;
SetBaseDatatypeReference();
TryMakeReferenceTo := TRUE;
END_METHOD

PROPERTY PUBLIC Value : ETcVnPixelPackMode
GET
Value := activeData;
END_GET
SET
activeData := Value;
END_SET
END_PROPERTY

END_FUNCTION_BLOCK

// ---- Datatypes/Aliases/_TcVnArray3_Point2_REAL.TcPOU
{attribute 'linkalways'} 
{attribute 'no_explicit_call' := 'This FB is a CLASS and must be accessed using methods or properties'}
{attribute 'enable_dynamic_creation'}
FUNCTION_BLOCK _TcVnArray3_Point2_REAL EXTENDS AliasDatatypeBase
VAR
	localData : TcVnArray3_Point2_REAL;
	activeData : REFERENCE TO TcVnArray3_Point2_REAL REF= localData;
	aliasBaseDatatype : _Array0to2OfTcVnPoint2_REAL;
END_VAR

PROPERTY PUBLIC Address : PVOID
GET
Address := ADR(activeData);
END_GET
END_PROPERTY

METHOD PUBLIC ClearReference
VAR_INPUT
END_VAR
activeData REF= localData;
SetBaseDatatypeReference();
END_METHOD

METHOD PUBLIC Clone : I_Datatype
VAR
    pClone : POINTER TO _TcVnArray3_Point2_REAL;
END_VAR
pClone := __NEW(_TcVnArray3_Point2_REAL);
Clone := pClone^;
END_METHOD

METHOD FB_init : BOOL
VAR_INPUT
	bInitRetains : BOOL; // if TRUE, the retain variables are initialized (warm start / cold start)
	bInCopyCode : BOOL;  // if TRUE, the instance afterwards gets moved into the copy code (online change)
	//InitialValue : TcVnArray4_LREAL; // if possible, not all values can be initialized
END_VAR
//localData := InitialValue; // if possible, not all values can be initialized
SetBaseDatatypeReference();
AddBaseDatatype(aliasBaseDatatype);
END_METHOD

PROPERTY PUBLIC Identifier : T_MAXSTRING
GET
Identifier := 'TcVnArray3_Point2_REAL';
END_GET
END_PROPERTY

METHOD PUBLIC MakeReferenceTo
VAR_INPUT
	ReferenceTarget : REFERENCE TO TcVnArray3_Point2_REAL;
END_VAR
activeData REF= ReferenceTarget;
SetBaseDatatypeReference();
END_METHOD

METHOD PROTECTED SetBaseDatatypeReference
VAR_INPUT
END_VAR
aliasBaseDatatype.MakeReferenceTo(activeData);
END_METHOD

PROPERTY PUBLIC Size : UDINT
GET
Size := SIZEOF(activeData);
END_GET
END_PROPERTY

METHOD TryMakeReferenceTo : BOOL
VAR_INPUT
	Target : I_Datatype;
END_VAR
VAR
	pTargetData : POINTER TO TcVnArray3_Point2_REAL;
END_VAR
IF NOT IsEquivalentTo(Target) THEN
	RETURN;
END_IF

pTargetData := Target.Address;
activeData REF= pTargetData^;
SetBaseDatatypeReference();
TryMakeReferenceTo := TRUE;
END_METHOD

PROPERTY PUBLIC Value : REFERENCE TO TcVnArray3_Point2_REAL
GET
Value REF= activeData;
END_GET
END_PROPERTY

END_FUNCTION_BLOCK

// ---- Datatypes/Arrays/_Array0to2OfTcVnPoint2_REAL.TcPOU
{attribute 'linkalways'} 
{attribute 'no_explicit_call' := 'This FB is a CLASS and must be accessed using methods or properties'}
{attribute 'enable_dynamic_creation'}
FUNCTION_BLOCK _Array0to2OfTcVnPoint2_REAL EXTENDS ArrayDatatypeBase_1D
VAR CONSTANT
	lBound : DINT := 0;
	uBound : DINT := 2;
END_VAR
VAR
	localData : ARRAY [lBound..uBound] OF TcVnPoint2_REAL;
	activeData : REFERENCE TO ARRAY [lBound..uBound] OF TcVnPoint2_REAL REF= localData;
	elements : ARRAY [lBound..uBound] OF _TcVnPoint2_REAL;
	baseType : _TcVnPoint2_REAL;
END_VAR

PROPERTY PUBLIC Address : PVOID
GET
Address := ADR(activeData);
END_GET
END_PROPERTY

PROPERTY PUBLIC BaseDatatype : I_Datatype
GET
BaseDatatype := baseType;
END_GET
END_PROPERTY

METHOD PUBLIC ClearReference
VAR_INPUT
END_VAR
activeData REF= localData;
SetElementReference();
END_METHOD

METHOD PUBLIC Clone : I_Datatype
VAR
    pClone : POINTER TO _Array0to2OfTcVnPoint2_REAL;
END_VAR
pClone := __NEW(_Array0to2OfTcVnPoint2_REAL());
pClone^.Value := Value;
Clone := pClone^;
END_METHOD

METHOD FB_init : BOOL
VAR_INPUT
	bInitRetains : BOOL; // if TRUE, the retain variables are initialized (warm start / cold start)
	bInCopyCode : BOOL;  // if TRUE, the instance afterwards gets moved into the copy code (online change)
END_VAR
SetElementReference();
END_METHOD

METHOD PUBLIC MakeReferenceTo
VAR_INPUT
	ReferenceTarget : REFERENCE TO ARRAY [lBound..uBound] OF TcVnPoint2_REAL;
END_VAR
activeData REF= ReferenceTarget;
SetElementReference();
END_METHOD

METHOD PROTECTED OnSerializeArrayValues
VAR_INPUT
	Serializer : I_Serializer;
END_VAR
VAR
	i : DINT;
END_VAR
FOR i := lBound TO uBound DO
	elements[i].SerializeWith(Serializer);
END_FOR
END_METHOD

METHOD PROTECTED SetElementReference
VAR_INPUT
END_VAR
VAR
	i : DINT;
END_VAR
FOR i := lBound TO uBound DO
	elements[i].MakeReferenceTo(activeData[i]);
END_FOR
END_METHOD

PROPERTY PUBLIC Size : UDINT
GET
Size := SIZEOF(activeData);
END_GET
END_PROPERTY

METHOD PROTECTED TryDeserializeArrayValues : BOOL
VAR_INPUT
	Deserializer : I_Deserializer;
	Feedback : I_DeserializerFeedback;
END_VAR
VAR
	enumerator : I_DeserializerArrayForwardEnumerator;
	i : DINT;
END_VAR
enumerator := Deserializer.GetArrayEnumerator();
i := lBound;

WHILE enumerator.MoveNext() AND i <= uBound DO
	
	IF NOT elements[i].TryDeserializeFrom(enumerator.Current, Feedback) THEN
		EXIT;
	END_IF
	i := i + 1;

END_WHILE
enumerator.Dispose();
END_METHOD

METHOD PUBLIC TryGetElementAsDatatypeByIndex : BOOL
VAR_INPUT
	Index : DINT;
	Destination : REFERENCE TO I_Datatype;
END_VAR
IF Index < lbound OR Index > ubound THEN
	RETURN;
END_IF

Destination := elements[Index];
TryGetElementAsDatatypeByIndex := TRUE;
END_METHOD

METHOD PUBLIC TryGetLowerBound : BOOL
VAR_INPUT
	Dimention : UDINT;
	Destination : REFERENCE TO DINT;
END_VAR
IF Dimention = 1 THEN
	Destination := lBound;
	TryGetLowerBound := TRUE;
END_IF
END_METHOD

METHOD PUBLIC TryGetUpperBound : BOOL
VAR_INPUT
	Dimention : UDINT;
	Destination : REFERENCE TO DINT;
END_VAR
IF Dimention = 1 THEN
	Destination := uBound;
	TryGetUpperBound := TRUE;
END_IF
END_METHOD

METHOD TryMakeReferenceTo : BOOL
VAR_INPUT
	Target : I_Datatype;
END_VAR
VAR
	pTargetData : POINTER TO ARRAY [lBound..uBound] OF TcVnPoint2_REAL;
END_VAR
IF NOT IsEquivalentTo(Target) THEN
	RETURN;
END_IF

pTargetData := Target.Address;
activeData REF= pTargetData^;
SetElementReference();
TryMakeReferenceTo := TRUE;
END_METHOD

PROPERTY PUBLIC Value : REFERENCE TO ARRAY [lBound..uBound] OF TcVnPoint2_REAL;
GET
Value ref= activeData;
END_GET
END_PROPERTY

END_FUNCTION_BLOCK

// ---- Datatypes/Aliases/_TcVnArray7_LREAL.TcPOU
{attribute 'linkalways'} 
{attribute 'no_explicit_call' := 'This FB is a CLASS and must be accessed using methods or properties'}
{attribute 'enable_dynamic_creation'}
FUNCTION_BLOCK _TcVnArray7_LREAL EXTENDS AliasDatatypeBase
VAR
	localData : TcVnArray7_LREAL;
	activeData : REFERENCE TO TcVnArray7_LREAL REF= localData;
	aliasBaseDatatype : _Array0to6OfLREAL;
END_VAR

PROPERTY PUBLIC Address : PVOID
GET
Address := ADR(activeData);
END_GET
END_PROPERTY

METHOD PUBLIC ClearReference
VAR_INPUT
END_VAR
activeData REF= localData;
SetBaseDatatypeReference();
END_METHOD

METHOD PUBLIC Clone : I_Datatype
VAR
    pClone : POINTER TO _TcVnArray7_LREAL;
END_VAR
pClone := __NEW(_TcVnArray7_LREAL);
Clone := pClone^;
END_METHOD

METHOD FB_init : BOOL
VAR_INPUT
	bInitRetains : BOOL; // if TRUE, the retain variables are initialized (warm start / cold start)
	bInCopyCode : BOOL;  // if TRUE, the instance afterwards gets moved into the copy code (online change)
	//InitialValue : TcVnArray7_LREAL; // if possible, not all values can be initialized
END_VAR
//localData := InitialValue; // if possible, not all values can be initialized
SetBaseDatatypeReference();
AddBaseDatatype(aliasBaseDatatype);
END_METHOD

PROPERTY PUBLIC Identifier : T_MAXSTRING
GET
Identifier := 'TcVnArray7_LREAL';
END_GET
END_PROPERTY

METHOD PUBLIC MakeReferenceTo
VAR_INPUT
	ReferenceTarget : REFERENCE TO TcVnArray7_LREAL;
END_VAR
activeData REF= ReferenceTarget;
SetBaseDatatypeReference();
END_METHOD

METHOD PROTECTED SetBaseDatatypeReference
VAR_INPUT
END_VAR
aliasBaseDatatype.MakeReferenceTo(activeData);
END_METHOD

PROPERTY PUBLIC Size : UDINT
GET
Size := SIZEOF(activeData);
END_GET
END_PROPERTY

METHOD TryMakeReferenceTo : BOOL
VAR_INPUT
	Target : I_Datatype;
END_VAR
VAR
	targetAsAlias : I_AliasDatatype;
	pTargetData : POINTER TO TcVnArray7_LREAL;
END_VAR
IF NOT Target.TryResolveAsAliasDatatype(targetAsAlias) THEN
	RETURN;
END_IF

IF targetAsAlias.Identifier <> Identifier THEN
	RETURN;
END_IF

pTargetData := Target.Address;
activeData REF= pTargetData^;
SetBaseDatatypeReference();
TryMakeReferenceTo := TRUE;
END_METHOD

PROPERTY PUBLIC Value : REFERENCE TO TcVnArray7_LREAL
GET
Value REF= activeData;
END_GET
END_PROPERTY

END_FUNCTION_BLOCK

// ---- Datatypes/Arrays/_Array0to6OfLREAL.TcPOU
{attribute 'linkalways'} 
{attribute 'no_explicit_call' := 'This FB is a CLASS and must be accessed using methods or properties'}
{attribute 'enable_dynamic_creation'}
FUNCTION_BLOCK _Array0to6OfLREAL EXTENDS ArrayDatatypeBase_1D
VAR CONSTANT
	lBound : DINT := 0;
	uBound : DINT := 6;
END_VAR
VAR
	localData : ARRAY [lBound..uBound] OF LREAL;
	activeData : REFERENCE TO ARRAY [lBound..uBound] OF LREAL REF= localData;
	elements : ARRAY [lBound..uBound] OF _LREAL(0.0);
	baseType : _LREAL(0.0);
END_VAR

PROPERTY PUBLIC Address : PVOID
GET
Address := ADR(activeData);
END_GET
END_PROPERTY

PROPERTY PUBLIC BaseDatatype : I_Datatype
GET
BaseDatatype := baseType;
END_GET
END_PROPERTY

METHOD PUBLIC ClearReference
VAR_INPUT
END_VAR
activeData REF= localData;
SetElementReference();
END_METHOD

METHOD PUBLIC Clone : I_Datatype
VAR
    pClone : POINTER TO _Array0to6OfLREAL;
END_VAR
pClone := __NEW(_Array0to6OfLREAL());
pClone^.Value := Value;
Clone := pClone^;
END_METHOD

METHOD FB_init : BOOL
VAR_INPUT
	bInitRetains : BOOL; // if TRUE, the retain variables are initialized (warm start / cold start)
	bInCopyCode : BOOL;  // if TRUE, the instance afterwards gets moved into the copy code (online change)
END_VAR
SetElementReference();
END_METHOD

METHOD PUBLIC MakeReferenceTo
VAR_INPUT
	ReferenceTarget : REFERENCE TO ARRAY [lBound..uBound] OF LREAL;
END_VAR
activeData REF= ReferenceTarget;
SetElementReference();
END_METHOD

METHOD PROTECTED OnSerializeArrayValues
VAR_INPUT
	Serializer : I_Serializer;
END_VAR
VAR
	i : DINT;
END_VAR
FOR i := lBound TO uBound DO
	elements[i].SerializeWith(Serializer);
END_FOR
END_METHOD

METHOD PROTECTED SetElementReference
VAR_INPUT
END_VAR
VAR
	i : DINT;
END_VAR
FOR i := lBound TO uBound DO
	elements[i].MakeReferenceTo(activeData[i]);
END_FOR
END_METHOD

PROPERTY PUBLIC Size : UDINT
GET
Size := SIZEOF(activeData);
END_GET
END_PROPERTY

METHOD PROTECTED TryDeserializeArrayValues : BOOL
VAR_INPUT
	Deserializer : I_Deserializer;
	Feedback : I_DeserializerFeedback;
END_VAR
VAR
	enumerator : I_DeserializerArrayForwardEnumerator;
	i : DINT;
END_VAR
enumerator := Deserializer.GetArrayEnumerator();
i := lBound;

WHILE enumerator.MoveNext() AND i <= uBound DO
	
	IF NOT elements[i].TryDeserializeFrom(enumerator.Current, Feedback) THEN
		EXIT;
	END_IF
	i := i + 1;

END_WHILE
enumerator.Dispose();
END_METHOD

METHOD PUBLIC TryGetElementAsDatatypeByIndex : BOOL
VAR_INPUT
	Index : DINT;
	Destination : REFERENCE TO I_Datatype;
END_VAR
IF Index < lbound OR Index > ubound THEN
	RETURN;
END_IF

Destination := elements[Index];
TryGetElementAsDatatypeByIndex := TRUE;
END_METHOD

METHOD PUBLIC TryGetLowerBound : BOOL
VAR_INPUT
	Dimention : UDINT;
	Destination : REFERENCE TO DINT;
END_VAR
IF Dimention = 1 THEN
	Destination := lBound;
	TryGetLowerBound := TRUE;
END_IF
END_METHOD

METHOD PUBLIC TryGetUpperBound : BOOL
VAR_INPUT
	Dimention : UDINT;
	Destination : REFERENCE TO DINT;
END_VAR
IF Dimention = 1 THEN
	Destination := uBound;
	TryGetUpperBound := TRUE;
END_IF
END_METHOD

METHOD TryMakeReferenceTo : BOOL
VAR_INPUT
	Target : I_Datatype;
END_VAR
VAR
	pTargetData : POINTER TO ARRAY [lBound..uBound] OF LREAL;
END_VAR
IF NOT IsEquivalentTo(Target) THEN
	RETURN;
END_IF

pTargetData := Target.Address;
activeData REF= pTargetData^;
SetElementReference();
TryMakeReferenceTo := TRUE;
END_METHOD

PROPERTY PUBLIC Value : REFERENCE TO ARRAY [lBound..uBound] OF LREAL;
GET
Value ref= activeData;
END_GET
END_PROPERTY

END_FUNCTION_BLOCK

// ---- Datatypes/Aliases/_TcVnArray8_LREAL.TcPOU
{attribute 'linkalways'} 
{attribute 'no_explicit_call' := 'This FB is a CLASS and must be accessed using methods or properties'}
{attribute 'enable_dynamic_creation'}
FUNCTION_BLOCK _TcVnArray8_LREAL EXTENDS AliasDatatypeBase
VAR
	localData : TcVnArray8_LREAL;
	activeData : REFERENCE TO TcVnArray8_LREAL REF= localData;
	aliasBaseDatatype : _Array0to7OfLREAL;
END_VAR

PROPERTY PUBLIC Address : PVOID
GET
Address := ADR(activeData);
END_GET
END_PROPERTY

METHOD PUBLIC ClearReference
VAR_INPUT
END_VAR
activeData REF= localData;
SetBaseDatatypeReference();
END_METHOD

METHOD PUBLIC Clone : I_Datatype
VAR
    pClone : POINTER TO _TcVnArray8_LREAL;
END_VAR
pClone := __NEW(_TcVnArray8_LREAL);
Clone := pClone^;
END_METHOD

METHOD FB_init : BOOL
VAR_INPUT
	bInitRetains : BOOL; // if TRUE, the retain variables are initialized (warm start / cold start)
	bInCopyCode : BOOL;  // if TRUE, the instance afterwards gets moved into the copy code (online change)
	//InitialValue : TcVnArray8_LREAL; // if possible, not all values can be initialized
END_VAR
//localData := InitialValue; // if possible, not all values can be initialized
SetBaseDatatypeReference();
AddBaseDatatype(aliasBaseDatatype);
END_METHOD

PROPERTY PUBLIC Identifier : T_MAXSTRING
GET
Identifier := 'TcVnArray8_LREAL';
END_GET
END_PROPERTY

METHOD PUBLIC MakeReferenceTo
VAR_INPUT
	ReferenceTarget : REFERENCE TO TcVnArray8_LREAL;
END_VAR
activeData REF= ReferenceTarget;
SetBaseDatatypeReference();
END_METHOD

METHOD PROTECTED SetBaseDatatypeReference
VAR_INPUT
END_VAR
aliasBaseDatatype.MakeReferenceTo(activeData);
END_METHOD

PROPERTY PUBLIC Size : UDINT
GET
Size := SIZEOF(activeData);
END_GET
END_PROPERTY

METHOD TryMakeReferenceTo : BOOL
VAR_INPUT
	Target : I_Datatype;
END_VAR
VAR
	targetAsAlias : I_AliasDatatype;
	pTargetData : POINTER TO TcVnArray8_LREAL;
END_VAR
IF NOT Target.TryResolveAsAliasDatatype(targetAsAlias) THEN
	RETURN;
END_IF

IF targetAsAlias.Identifier <> Identifier THEN
	RETURN;
END_IF

pTargetData := Target.Address;
activeData REF= pTargetData^;
SetBaseDatatypeReference();
TryMakeReferenceTo := TRUE;
END_METHOD

PROPERTY PUBLIC Value : REFERENCE TO TcVnArray8_LREAL
GET
Value REF= activeData;
END_GET
END_PROPERTY

END_FUNCTION_BLOCK

// ---- Datatypes/Arrays/_Array0to7OfLREAL.TcPOU
{attribute 'linkalways'} 
{attribute 'no_explicit_call' := 'This FB is a CLASS and must be accessed using methods or properties'}
{attribute 'enable_dynamic_creation'}
FUNCTION_BLOCK _Array0to7OfLREAL EXTENDS ArrayDatatypeBase_1D
VAR CONSTANT
	lBound : DINT := 0;
	uBound : DINT := 7;
END_VAR
VAR
	localData : ARRAY [lBound..uBound] OF LREAL;
	activeData : REFERENCE TO ARRAY [lBound..uBound] OF LREAL REF= localData;
	elements : ARRAY [lBound..uBound] OF _LREAL(0.0);
	baseType : _LREAL(0.0);
END_VAR

PROPERTY PUBLIC Address : PVOID
GET
Address := ADR(activeData);
END_GET
END_PROPERTY

PROPERTY PUBLIC BaseDatatype : I_Datatype
GET
BaseDatatype := baseType;
END_GET
END_PROPERTY

METHOD PUBLIC ClearReference
VAR_INPUT
END_VAR
activeData REF= localData;
SetElementReference();
END_METHOD

METHOD PUBLIC Clone : I_Datatype
VAR
    pClone : POINTER TO _Array0to7OfLREAL;
END_VAR
pClone := __NEW(_Array0to7OfLREAL());
pClone^.Value := Value;
Clone := pClone^;
END_METHOD

METHOD FB_init : BOOL
VAR_INPUT
	bInitRetains : BOOL; // if TRUE, the retain variables are initialized (warm start / cold start)
	bInCopyCode : BOOL;  // if TRUE, the instance afterwards gets moved into the copy code (online change)
END_VAR
SetElementReference();
END_METHOD

METHOD PUBLIC MakeReferenceTo
VAR_INPUT
	ReferenceTarget : REFERENCE TO ARRAY [lBound..uBound] OF LREAL;
END_VAR
activeData REF= ReferenceTarget;
SetElementReference();
END_METHOD

METHOD PROTECTED OnSerializeArrayValues
VAR_INPUT
	Serializer : I_Serializer;
END_VAR
VAR
	i : DINT;
END_VAR
FOR i := lBound TO uBound DO
	elements[i].SerializeWith(Serializer);
END_FOR
END_METHOD

METHOD PROTECTED SetElementReference
VAR_INPUT
END_VAR
VAR
	i : DINT;
END_VAR
FOR i := lBound TO uBound DO
	elements[i].MakeReferenceTo(activeData[i]);
END_FOR
END_METHOD

PROPERTY PUBLIC Size : UDINT
GET
Size := SIZEOF(activeData);
END_GET
END_PROPERTY

METHOD PROTECTED TryDeserializeArrayValues : BOOL
VAR_INPUT
	Deserializer : I_Deserializer;
	Feedback : I_DeserializerFeedback;
END_VAR
VAR
	enumerator : I_DeserializerArrayForwardEnumerator;
	i : DINT;
END_VAR
enumerator := Deserializer.GetArrayEnumerator();
i := lBound;

WHILE enumerator.MoveNext() AND i <= uBound DO
	
	IF NOT elements[i].TryDeserializeFrom(enumerator.Current, Feedback) THEN
		EXIT;
	END_IF
	i := i + 1;

END_WHILE
enumerator.Dispose();
END_METHOD

METHOD PUBLIC TryGetElementAsDatatypeByIndex : BOOL
VAR_INPUT
	Index : DINT;
	Destination : REFERENCE TO I_Datatype;
END_VAR
IF Index < lbound OR Index > ubound THEN
	RETURN;
END_IF

Destination := elements[Index];
TryGetElementAsDatatypeByIndex := TRUE;
END_METHOD

METHOD PUBLIC TryGetLowerBound : BOOL
VAR_INPUT
	Dimention : UDINT;
	Destination : REFERENCE TO DINT;
END_VAR
IF Dimention = 1 THEN
	Destination := lBound;
	TryGetLowerBound := TRUE;
END_IF
END_METHOD

